0.902067723111, 0.547746633735, 0.158435508917, -0.208265848525, -0.628990277088, 0.572162738409, 0.091285246118, 0.383730288054, 0.903400742168, 0.899370619505, 0.409534416843, 0.721432036419, -0.171166404881, 0.037531974106, -0.923997071504, -0.113982760314, -0.780465516076, -0.697778906118, 0.818445268006, -0.590523809214, -0.171407635527, -0.610750438511, -0.662726470352, 0.271639270079, 0.430827816825, -0.113990542861, 0.717940707740, 0.748908513575, 0.136771315412, 0.820956531665, -0.827648688243, -0.863989622980, 0.510781040232, -0.902120915451, -0.807354979352, -0.349421748268, 0.635400432082, -0.484592911038, -0.334974188576, -0.625415861932, -0.571767841976, -0.465300639249, -0.877974358194, -0.295243416993, 0.744226620731, -0.179565886893, 0.207531340996, -0.366675890084, -0.149096543674, -0.117815700724, 0.428201432730, -0.223791727240, -0.374806082459, -0.996388861807, -0.079249452770, -0.509844081507, -0.045674891403, -0.440046273099, -0.482288649525, 0.214892790090, -0.035347344465, -0.179260400766, -0.678074715747, -0.440784613352, 0.695462715044, 0.799643546103, 0.121836725671, -0.525839633185, 0.541538631258, 0.042687636792, 0.657176601005, 0.400032534671, 0.390034269384, -0.114184467168, 0.994123486006, 0.464706416014, -0.894852671561, -0.267108894190, 0.402002424630, 0.160977296129, 0.145466358788, 0.976531073927, 0.056719064699, -0.108518014803, 0.248657955733, 0.642098807478, 0.882274575211, -0.075050234752, -0.387849389007, 0.617082980694, 0.668408355761, -0.990995438959, -0.796071114181, 0.934107014787, -0.282962962945, 0.914221612194, -0.454371406874, 0.420398416529, -0.665824266955, -0.618566845789, 0.831084959587, -0.534987119828, 0.461148218286, 0.306078529549, -0.151742796527, -0.026015973197, -0.157735142413, -0.339520290351, -0.931051734632, -0.365346093645, -0.002225437347, 0.232831108132, -0.177404032820, 0.882245684523, -0.954178340038, 0.274990354804, -0.399527887776, 0.358048197887, 0.673515953803, 0.518411076586, -0.415020034931, -0.299868827720, 0.047456389550, 0.214993655963, 0.268555680928, -0.968453108577, 0.257861939024, 0.379408565827, 0.965913300373, -0.875854620537, 0.402543694330, -0.538524422114, -0.875649232985, -0.863428966901, -0.882617351428, 0.375087296705, 0.673440480300, 0.292068266375, 0.644043062216, -0.380148068958, -0.859870226482, -0.686025308272, -0.555657058657, -0.340355923972, -0.657490223017, 0.568129117819, 0.872158742728, 0.670356628639, -0.477574660769, 0.817331344706, -0.679945936582, 0.915722789645, 0.046172274302, 0.637048459704, 0.820068547051, 0.613851939895, 0.523961727584, -0.231042052914, 0.685545054075, 0.038349575245, 0.401627308689, -0.165043382722, -0.476005923500, 0.181897513589, -0.509728059258, 0.711934265898, -0.110910195960, 0.135544444946, -0.203545678322, 0.121725756239, 0.667875415090, -0.662629857099, 0.534453835551, 0.073534356101, 0.955674602016, 0.716327577401, -0.505383061461, 0.201464649072, -0.255533045943, -0.628786980533, -0.588780931270, -0.186636679105, -0.899471910220, 0.637859966244, -0.685918583844, 0.751607301602, 0.823050845274, 0.874034840312, 0.350531785053, 0.364133563102, 0.417303337627, -0.759031868112, -0.159714839585, -0.572495224891, 0.683268462042, -0.476691720750, 0.867949662476, -0.986907373894, -0.195229753954, 0.446764162700, -0.007593856855, -0.385917986662, -0.999910422090, -0.288038894845, 0.247883233370, 0.499214163589, -0.979960644666, 0.409109548152, 0.604365030955, -0.752059503253, -0.098716987436, 0.261840857748, -0.310421840836, 0.273036546583, 0.966283042994, -0.512419815859, 0.223807017157, 0.204832588236, -0.126778911159, 0.559677233312, -0.312489754796, -0.130559768854, 0.344979245612, -0.995738541041, 0.850135154641, 0.859556583783, -0.543090391431, 0.363764893193, 0.863579500924, 0.416769655519, -0.716493357372, 0.165233723667, 0.879255846651, -0.719193755109, 0.827530877332, 0.296285159044, 0.257581488476, 0.429469163603, -0.296730775590, -0.247378135775, -0.475968969101, 0.156990696039, -0.110782913209, -0.397894591632, 0.928031296231, 0.820762403773, -0.777284120923, 0.829749477105, -0.225872893277, 0.521154183131, -0.448414615240, -0.107872120866, -0.839344971377, -0.477732735712, 0.067316773398, 0.269758615907, 0.052404674492, -0.967008085228, -0.077971909436, -0.832627790185, -0.897211929296, -0.750780680221, 0.148919714675, 0.064021695691, 0.427457969280, -0.064800288486, 0.247754925621, -0.612484958621, 0.875249801105, 0.647953509070, -0.259754750240, -0.368335454917, 0.636967637997, -0.656662520290, -0.097478340411, -0.837053812543, 0.527496448987, -0.501134811721, -0.031980809441, -0.889659422432, -0.729835289653, -0.403920662593, 0.911833319274, -0.195394608538, 0.579983597887, 0.480878402094, 0.753295698404, -0.886557102388, -0.481051881669, 0.858752026661, 0.419439422595, 0.424707540380, 0.070671397664, -0.607165311260, -0.423632073663, 0.067909420480, -0.598470181812, -0.525774866523, 0.950714625230, 0.599861469287, -0.442861591818, 0.069620972834, 0.541300442667, 0.327490730799, 0.309082582040, 0.047253630814, 0.606651953953, 0.112544392696, 0.218055864524, 0.106968569698, 0.599462743203, 0.023550831903, 0.337815059310, 0.932264427175, 0.165960823492, 0.733249781045, -0.789431880042, 0.493722751772, -0.004488036016, -0.691545281081, 0.051434132048, -0.767664479342, 0.141488503409, -0.281316569424, -0.517286821248, 0.770675414438, 0.853427796276, -0.657209527482, -0.742725530343, -0.427013088695, -0.483223026887, 0.856541610703, 0.723705297730, -0.817544392274, -0.863812634951, 0.190487237743, 0.462198474418, 0.038100294980, 0.386360398109, 0.138093633863, 0.668065694067, -0.322052819469, 0.694404971202, 0.497259150758, 0.048078271919, 0.614850342950, -0.443216140498, -0.793653679765, 0.901627621897, 0.311872553282, 0.787310048058, -0.793855935575, -0.913720147731, -0.322313905779, -0.139500835847, -0.031831499233, -0.199892750670, 0.779717894037, 0.221123175177, -0.472991991045, 0.820421631406, -0.784247416860, -0.382988401296, -0.862138590325, 0.423435170567, -0.804372214538, -0.876593305913, 0.414554638112, 0.690384876731, -0.460644141012, -0.473321310585, -0.262625983811, 0.898335619536, 0.260679529821, 0.275699048997, -0.994264328699, 0.602960163802, -0.216638281855, -0.490344920037, 0.737015766298, 0.221647194511, -0.352968279409, -0.134519186654, -0.273626093464, 0.709228485444, -0.663208857573, -0.757535911133, 0.918108741001, -0.942949058606, 0.684475031813, -0.682159656169, 0.044424281903, -0.681026442177, -0.550846721858, 0.680676646566, 0.115083908438, -0.475380034855, 0.031236674021, 0.309528795181, 0.396497086310, 0.992561703820, -0.828608440171, -0.662821048169, 0.345443857269, 0.511783158770, 0.701092811961, -0.154665388649, 0.857411359782, 0.807768488786, 0.176563276807, -0.262657388798, -0.537263630008, 0.327682125245, -0.195002137162, 0.416130858898, -0.466182630628, 0.440430297927, -0.558656953019, -0.133970113749, 0.877224542781, -0.640643669335, 0.175780660046, -0.147882721452, 0.214081434003, 0.055607726695, -0.504690715015, -0.647660320770, 0.141522624346, -0.709032275134, 0.560486701112, -0.692619269210, -0.323622492407, -0.856721228447, 0.538047401446, -0.385786684720, 0.497652128026, -0.608579764541, 0.046673550854, -0.524716032653, -0.513458687505, -0.802148264126, -0.718972019465, -0.809695136345, -0.174937573729, -0.459699622109, -0.431556777774, -0.377164596626, -0.653806773416, -0.495328156416, -0.376523729440, 0.669045504275, 0.687682292995, 0.409745264703, 0.409698822451, -0.314637937582, 0.421181934329, 0.426145288987, 0.411239972315, -0.143971067142, -0.472530929786, -0.999376532103, -0.010117384944, -0.252446404507, 0.568689736131, -0.384579797806, 0.105797046275, -0.986014968661, -0.358988842273, 0.463099585531, 0.579498127847, 0.174069383888, -0.294564146505, 0.383791518921, -0.352819525007, -0.751197789421, 0.238384371689, 0.575958789292, 0.325567966100, -0.775702038994, 0.586055162359, 0.015762489652, -0.790104117329, 0.105873643257, 0.411658492741, -0.348339320392, -0.982719945801, 0.548902146145, -0.825606404302, 0.197116056386, -0.658666172336, -0.964479301316, -0.818704439072, -0.644408803838, -0.578548088605, -0.925692159326, -0.228069188766, -0.662552251899, 0.145382647632, 0.410827400040, -0.097163171197, 0.524975835549, -0.545350325804, -0.924369765877, -0.871078875314, 0.640834814893, 0.745794714895, 0.645476673311, 0.816373640524, 0.660481824045, -0.019329983308, -0.174444134561, 0.008509437553, 0.718182955315, 0.421438827594, -0.589750350198, 0.863020074421, -0.534470850901, -0.487310067966, -0.046868309168, 0.118498474737, -0.567631551457, -0.893789349031, 0.111917085452, -0.780230280061, -0.653497496174, 0.517018493288, 0.220633771232, 0.459112770183, -0.928205266632, 0.656898353644, -0.483808580172, 0.547447574349, -0.674440746574, -0.610672731793, 0.927277458029, 0.825506128691, 0.248231844156, -0.478557259882, 0.670298284369, -0.043719508526, -0.290727658337, -0.361422090257, 0.948970050555, 0.571211060537, 0.331947663435, 0.391540362592, -0.168129930820, 0.788132594964, -0.458071788013, -0.057843938125, -0.615253173260, 0.299805842239, -0.802359906586, -0.271655375124, -0.583424020451, 0.247170669845, -0.089237113690, -0.955580797901, -0.691849111829, -0.625525753810, 0.334321355052, -0.210250415701, 0.975713460950, -0.551570788964, -0.735481025987, -0.576053802898, -0.437960036849, 0.322455075861, 0.309870803261, -0.316773385043, 0.928040673837, -0.121478860441, 0.936985092037, 0.334479511865, 0.077340483645, 0.804023797725, -0.260543885714, 0.352038790026, -0.673334760316, -0.577768216694, 0.092893685951, 0.211080078462, 0.404319179727, -0.249737852186, 0.752486932045, 0.162398853086, -0.901051886249, 0.486410134054, -0.979809914914, -0.198115550586, -0.007249442145, 0.797872230895, 0.997717591935, 0.732814017231, 0.892591137252, 0.498196079629, -0.815816982001, -0.050342233270, -0.521236123169, -0.349672510594, 0.132732176530, 0.892460200155, -0.751690695745, 0.645648352953, 0.295298566529, 0.596168128515, 0.753852190381, 0.775889617173, 0.599280300543, 0.768789926120, -0.095563371426, -0.973844451721, 0.524080710421, -0.376303503006, -0.485229695550, -0.858942355628, 0.500599253436, 0.039926936378, -0.449610628307, 0.124016399453, 0.555638716739, -0.498417758413, -0.420856983175, 0.999029911090, -0.961093982264, -0.738289444812, -0.085192780626, 0.391810947010, 0.516447957312, -0.639465369036, -0.837091914030, 0.699360516292, -0.198587431368, 0.082410681736, 0.765720099984, -0.177359173445, -0.031876021494, -0.479541180246, -0.740542530919, 0.957917378801, -0.948390493476, 0.866574505446, 0.093655648830, -0.944034261871, 0.773327126883, -0.574295769670, -0.518124168627, 0.293613250173, -0.597473245068, 0.755945496046, 0.933304784644, -0.333019192500, 0.383238400688, 0.526374353051, -0.853584808087, -0.738580426032, -0.331110505691, 0.524178678541, -0.495558182949, -0.899076756135, -0.015412120276, -0.092582756823, 0.697556773482, -0.499966619988, -0.036853902291, 0.879312708384, -0.109576945084, 0.009175009685, 0.099508293099, 0.136935455562, 0.392722695828, -0.420667048584, 0.607127244576, 0.984695379888, -0.163782934507, -0.549644422923, 0.513549503570, 0.925508393581, -0.255009979572, 0.609262841823, -0.021193500239, -0.541789592832, -0.613882790944, 0.902155639323, 0.678615981560, -0.461929508006, -0.084629200065, -0.273007190663, -0.711194393717, 0.499258514395, 0.625397679928, 0.664594211938, -0.263197178606, 0.620762842919, 0.882348542333, 0.928022772401, -0.334853145062, -0.154845691010, 0.863815493458, -0.829639009837, -0.182445739571, -0.906220219477, -0.561447714123, -0.769955136566, -0.594628431961, -0.292206696676, 0.618906581605, -0.439095465100, -0.366018131382, 0.407319088052, 0.732119312417, -0.735010247830, 0.678585596261, 0.339466473956, -0.881390338206, -0.736278151056, -0.889597356662, 0.541355736658, 0.316292775127, 0.148014392068, 0.223189988951, 0.479998607985, 0.330481521753, -0.223134566617, -0.190247914778, 0.281426168014, -0.296369895074, 0.718651766283, 0.869352765614, -0.207686781396, -0.782552643117, -0.651847670081, 0.455603345239, -0.488226839721, 0.163136971340, 0.800684569232, 0.858983058975, 0.751860753472, -0.358023298280, 0.325330482061, 0.809609122319, -0.760890582618, -0.928166736771, 0.656476871327, -0.937213106465, -0.921733664164, -0.475830893424, 0.508808172470, 0.255159840161, 0.259757582636, 0.705652729884, -0.087020950922, 0.976219451336, -0.355676086581, -0.936709635622, -0.979396294829, -0.898245320689, 0.596830327285, -0.217465147476, 0.228593853339, -0.788546553797, -0.896188841735, 0.710079375577, 0.834342165163, 0.194208097690, -0.889414160808, 0.627466473747, 0.448861767538, -0.889430622862, 0.729848135279, 0.232207840916, 0.678984740434, 0.513067189590, -0.364461172605, 0.900225308282, 0.898129693826, 0.388100392626, 0.675049186773, -0.496830148112, -0.246389044291, 0.422409485521, -0.069758471918, 0.282857299873, -0.097240820592, -0.713936274675, -0.411823071316, 0.572501368105, 0.389956703715, -0.758606826908, -0.127168931917, -0.850887781955, -0.554966871724, 0.894983424125, 0.185523938233, 0.693138358146, -0.197265191790, -0.203491160721, -0.972953478271, -0.776174524959, -0.789994922894, -0.302125475591, 0.366567086152, 0.696668458460, -0.262059911455, -0.091538051390, -0.174227813118, -0.521944029812, -0.639116745209, -0.994722702071, 0.248421896079, 0.733717564205, -0.441311340158, 0.768425722051, 0.520003199325, -0.639212138637, -0.180891064374, 0.519298301347, 0.180855598097, -0.612161679453, 0.754579307788, 0.960201120260, -0.476694950357, 0.637902991314, -0.883802242767, -0.406907694780, -0.698293447577, 0.363727624772, -0.551344329860, -0.789311971844, 0.611764313057, -0.933333158754, -0.816922461754, 0.152316955752, 0.478475923833, 0.955835157038, -0.992696367872, -0.215975653150, -0.596853601993, 0.175098734181, 0.291837294588, -0.349292385654, 0.491399179262, -0.353079439055, -0.590957321614, -0.874754887564, -0.961757632136, -0.930999458820, 0.283424173409, 0.520624351676, 0.008262324147, 0.020881745513, 0.744737608930, -0.679884618745, -0.831962244377, -0.840784651246, -0.560567109129, -0.642876168801, 0.311818897047, 0.101128681392, -0.638011814338, 0.872795850402, -0.159183999846, -0.904681946102, 0.354905173733, -0.515267683312, 0.581969072983, -0.127418089591, 0.230260937261, -0.741946939285, -0.200768179343, -0.980609810479, -0.684763731473, -0.516433875085, 0.986685959321, 0.470386428852, -0.872768208249, -0.558895352344, 0.149937150206, 0.615825539633, -0.264722417196, -0.377096516585, -0.856346137153, -0.788942459577, -0.870140315556, 0.163941326587, -0.404932474401, -0.086969831256, 0.275572447356, 0.130528653947, 0.225626064900, -0.300687807258, -0.063137772755, 0.413460969163, 0.430496368348, 0.374608436244, 0.110159988194, 0.383531273735, 0.026336885273, 0.481870944866, 0.572793544103, -0.841410923094, 0.726230130592, 0.422626465773, 0.987040902479, -0.752527232920, 0.337336279758, -0.274087008168, -0.005517808787, -0.921366596279, 0.916932265906, -0.497163751751, -0.155037225965, 0.310010659139, -0.566412550499, -0.275858488149, 0.510696795999, 0.823895828606, -0.598537121361, 0.481641736745, -0.435667888216, -0.412970162287, 0.453096732529, -0.750004660313, 0.121717794140, -0.720106880497, 0.432886094516, -0.074623212176, -0.020748418849, -0.078484791591, 0.636717008777, -0.067284118653, 0.375459220207, 0.124895765900, 0.230410446731, -0.902714563247, -0.001864722325, 0.937479300039, -0.131320027758, 0.841670010406, -0.968851784224, -0.184493168388, 0.905435162382, 0.692667741964, -0.317444067630, -0.722457782211, -0.739143464615, 0.035789919223, 0.068841841490, 0.511247473820, 0.322821098972, -0.212686382587, -0.007510391113, -0.487271832184, 0.949211182090, -0.307437882377, 0.449499244891, 0.162254494902, -0.306795679625, -0.010127440304, 0.747336956906, 0.142761180780, -0.640301590947, 0.531098984791, -0.857075049402, 0.663637731926, 0.817908313858, 0.878376984735, 0.797160005317, -0.408351772023, -0.784646267207, -0.780465634731, -0.676144467590, -0.610308003312, 0.844588028061, 0.829858125174, 0.643585446652, -0.426313608940, 0.399038497650, -0.164260528142, 0.997434039516, -0.641906502219, 0.208004147838, -0.440246526744, -0.603319814376, -0.697535413795, -0.915244348141, 0.023402903934, -0.615366330865, -0.949611352494, 0.563554375640, -0.871067117361, -0.832000580396, 0.897450898736, 0.126694941714, 0.027490221083, 0.495037617696, -0.836886933588, -0.536122764534, -0.369049545039, 0.180840357339, 0.578901094828, 0.173752573076, 0.952523280192, 0.685589076436, -0.588390745007, 0.584014422739, 0.389192578675, 0.805180913453, -0.837683150684, -0.535902970417, -0.795579368694, -0.672488921187, -0.401967403023, -0.266015411193, -0.700071656406, -0.661537605497, 0.428578951305, 0.307438231288, -0.319134311558, -0.158229865472, 0.122100948536, 0.316647537089, 0.654881180467, -0.601247643044, -0.285971434096, -0.120996636816, 0.307013345399, 0.024607912723, 0.780866321402, 0.827011782153, -0.408099091611, 0.278959308761, -0.324110908146, 0.954667413246, -0.994200123295, 0.733667119162, 0.982355521575, 0.585910600089, -0.245053104507, -0.869890049586, 0.390384356232, 0.055915341397, -0.494593369296, 0.067978157636, -0.209797929688, -0.234475593468, 0.097162281058, 0.870141800427, 0.096384253332, -0.952188287095, -0.731345573698, -0.165482635994, -0.187444199891, -0.591497502129, 0.332033942900, -0.690309656181, -0.396239220922, -0.156037720211, -0.215056180847, -0.769707059926, 0.675887223483, -0.906017205847, 0.876468187997, -0.708124183046, -0.281495100912, 0.776569334970, 0.857072888627, -0.809628008201, -0.079249219029, 0.406455587530, 0.627005649405, -0.155311231490, -0.857086400652, 0.274471601053, -0.930818098687, 0.007788139760, 0.465969417580, -0.416164815180, 0.992546790862, 0.993396258669, -0.012690712410, 0.938815587371, 0.010082268904, 0.333626233432, -0.946598206468, 0.023833684820, 0.755018710801, -0.583796230848, 0.744636654121, -0.054803308345, 0.119361100535, 0.904737230522, 0.105433415228, -0.100465796471, -0.400813965188, 0.986573964897, 0.960560568472, 0.343893558841, 0.321191542146, 0.591949840905, 0.203709843240, -0.089766909462, 0.659283434562, 0.834650680409, 0.599946686403, -0.893671061764, 0.185193125906, 0.598243851156, 0.494653358191, -0.824234498133, 0.330137485214, 0.459199718746, -0.380078786452, 0.621342974535, -0.201678517679, -0.585751577309, 0.352290586741, -0.669451432036, -0.218928073481, 0.058108217223, -0.031196588873, 0.092125031325, 0.346035679807, 0.623253353818, 0.833640879585, 0.090154576628, -0.377337664102, 0.558057164890, 0.281314752040, -0.033178260345, 0.759655753140, 0.133419436721, -0.007246190471, 0.375981724986, 0.185416510648, 0.445840061143, -0.598456736854, -0.273561798910, 0.635935834108, -0.671850717339, -0.183411776600, 0.656991651101, 0.282871652770, 0.685120867775, 0.166078367253, -0.264592070327, 0.542095741840, -0.519628703952, 0.500120307237, 0.741991020344, 0.255474688638, 0.918802912911, 0.199181168394, -0.594989788846, -0.571215380403, 0.608282066309, 0.460729143748, 0.833252717266, 0.084964647411, -0.370913351739, -0.363003122658, -0.925953646722, -0.782427060836, 0.846933504079, 0.285436644766, -0.143414031599, 0.668915138352, 0.898862442394, -0.437177081853, -0.179762632112, 0.483008894533, 0.574112519179, -0.282132247853, -0.671290005477, 0.182962117500, -0.500901080645, -0.131995091164, -0.008479864088, 0.570597108055, -0.522285784494, -0.698203600301, 0.567216683405, -0.253991031154, 0.198616690912, -0.206159691877, 0.874299254920, 0.916073463883, -0.177599802708, 0.052856943129, 0.321599342233, 0.487713571286, 0.434875109480, 0.454981547059, -0.447310547138, -0.751544863139, 0.257341399761, 0.738761982079, -0.915505782082, 0.918820821766, 0.489762818442, 0.108751866942, -0.142419326852, 0.045553815659, -0.053248908496, 0.564844001614, 0.576431440231, 0.197238681554, -0.554588211541, -0.896750490750, -0.107015089260, 0.757671946286, -0.988318593464, -0.285849613744, -0.070193964846, -0.866073238372, -0.131218499251, -0.542815144688, -0.192486590434, -0.104898053726, 0.403113899086, -0.350540387012, -0.915667517803, -0.332927497451, -0.335765375710, 0.038520578308, -0.143795935176, 0.441189786120, 0.650084443526, -0.656768821387, 0.723359834066, 0.828551591458, 0.308912870497, 0.676796020016, 0.065360105395, -0.922536305931, -0.348531898237, -0.513304823627, -0.297827637166, -0.082461528155, 0.016276713804, -0.786380409409, 0.678030100136, 0.147740819944, 0.176282510828, -0.431260850842, -0.132132095003, -0.413929670555, -0.005764474600, -0.330964537867, -0.100162800351, -0.472941169805, -0.542679986802, -0.874061105223, 0.100356010592, -0.463659755249, -0.278680910166, -0.542046476870, 0.552864273666, 0.468671758513, -0.124295035719, -0.460734974844, 0.668283199659, 0.927737905991, -0.167147762855, -0.277013105851, -0.923891595109, 0.906674795184, -0.455028116401, -0.540008041009, -0.494869166885, 0.526172181884, 0.109719054742, 0.081916195555, 0.388724821274, -0.476841311760, -0.937955600408, -0.595912447157, 0.832559243544, -0.899913786612, -0.276283055448, 0.506865544814, -0.407856026634, 0.615870788700, 0.275574874856, 0.450884058482, -0.913986586630, -0.349312684610, -0.030949128255, -0.719515909072, 0.665314379703, -0.154128193046, -0.371970584890, -0.621737057084, -0.723639193437, 0.950174798983, 0.003496887784, 0.863738081479, 0.063604209810, -0.344069899287, -0.837636455085, -0.277143252239, 0.179692395755, -0.399215308999, 0.650553170401, 0.047417792552, 0.053148296668, 0.659544150477, 0.432211420512, -0.281196656581, 0.667557712592, -0.671350631398, -0.236148780578, 0.956216656540, 0.817977570264, 0.427997328548, -0.155470437325, 0.519823354454, -0.268595554176, 0.006613729587, -0.803166393168, 0.305451800563, 0.625532453949, -0.611482469379, 0.041672018585, 0.175701108134, -0.932207163341, -0.570526755069, -0.182547074452, 0.208498231301, 0.361165944766, 0.413513154068, 0.401338295736, 0.407815956316, -0.467221204260, 0.644252080100, -0.091443607103, 0.957892815619, -0.440636580169, -0.387089664734, -0.493075638781, 0.641286876349, -0.028253600635, 0.580984483796, -0.692302690704, 0.113217917648, 0.090548988898, 0.285623446365, -0.913546296501, 0.288219985462, 0.615633782362, -0.778091071411, -0.431404256373, 0.909327872495, 0.827143535825, 0.545499754688, 0.134469798778, -0.669786232709, -0.937669371482, -0.558688270138, -0.116439050790, -0.372460446644, 0.555591598562, -0.960017793317, -0.746107610008, 0.511851771589, -0.365835468561, 0.707396975177, -0.019130076624, -0.602736726515, -0.458292025987, 0.315853928913, 0.385721257797, -0.175073250788, 0.485108885409, 0.263458181878, 0.282884209581, 0.252253570847, -0.885262243135, -0.901965958264, -0.586618336778, 0.586978002277, 0.956268688056, -0.026652825884, 0.526689044036, 0.084461592036, 0.992199164064, -0.046696321528, -0.204073634724, -0.572075186271, 0.667129135406, -0.557670840681, -0.623571944409, -0.127764794039, 0.677436036029, -0.243928992779, 0.115454645247, -0.106261316465, 0.875817640192, -0.911659216030, -0.723180445731, -0.749917607226, -0.143613217245, 0.510782846208, 0.592148535170, 0.755937850729, 0.143577208851, 0.748608641766, -0.047832373406, -0.277641989027, -0.393798066807, 0.906563806375, 0.236514075822, -0.654547536639, -0.547004015725, 0.319959414204, 0.810180401437, -0.492599210717, -0.642312728580, 0.563847564487, -0.429612325808, -0.905112594777, -0.952594002848, -0.346697424472, 0.583233488458, 0.073636746695, -0.136441075915, 0.082907096557, -0.305054636901, 0.285293010300, -0.893563847112, 0.322084070962, 0.971882025856, -0.146156755466, -0.356956540131, -0.746482271441, -0.309283733816, 0.651656064463, 0.375318446725, -0.431665101072, 0.619496901793, -0.702714202971, 0.213112447858, -0.454193434429, -0.076761482572, 0.977784305799, 0.275252647113, -0.846696395746, -0.797319732120, 0.372925045161, -0.772170292448, 0.640181446660, -0.380250960008, -0.287290543455, 0.224505263591, 0.011578759763, 0.944558001616, 0.806593283333, 0.515954696930, 0.084951472458, -0.316884986536, -0.864354010116, -0.003443897138, -0.690827655473, -0.008520744446, 0.220396687009, 0.200235831171, 0.685889373916, -0.014026315761, -0.787443790026, -0.907284922892, 0.939170388381, 0.925558380706, 0.161408122255, -0.044713406894, -0.394265986689, 0.379484965817, 0.014114186380, -0.623414619773, 0.817012000225, 0.255261319168, 0.135582969896, 0.338465737203, 0.442524817903, -0.466978297911, -0.168652193127, -0.151517063576, -0.358379111216, 0.643324049335, -0.085836757439, 0.340949770070, -0.245096435721, -0.799980577993, -0.764459273351, 0.467513495684, 0.783026918621, -0.637839056728, 0.445638069827, -0.263730123257, 0.010592797117, -0.679534831443, 0.021620059157, 0.194340703903, 0.113573130237, 0.784868487428, -0.149437997084, -0.204534660833, 0.927329646419, -0.644591449821, -0.852819168526, 0.473848525185, 0.126952720835, 0.899645866835, 0.893068661739, -0.319139968905, -0.018704087532, -0.988755218068, -0.944404487873, -0.658413493227, 0.120834469199, 0.602879864628, -0.776891717498, -0.062369291396, 0.873428958418, -0.784975379154, -0.846081915762, -0.142634809539, 0.931194504200, -0.313697070642, 0.305513351038, 0.257762908231, -0.927682360219, -0.098896303981, 0.874223085823, -0.537347706236, 0.803169888173, 0.488848844625, 0.382007913398, 0.964750985250, -0.758298724618, 0.537455786487, 0.107640861046, 0.544733170083, 0.868079577869, 0.948820240533, -0.216135578088, -0.698443512442, 0.523734529075, -0.833728868662, -0.238937528073, -0.965614216705, 0.974503056657, -0.449732043573, -0.816792244667, 0.473488661445, 0.538573132000, 0.927032186378, -0.015042549161, 0.900491473952, 0.744018480803, -0.160571460367, 0.347232615524, -0.740895859057, 0.597252212874, 0.398417747784, 0.232333936277, 0.649709894456, -0.925999495066, 0.208587663975, 0.022625988947, -0.717523335040, 0.528684482541, -0.675050725574, -0.935182112512, 0.885518136690, -0.482580827497, -0.307067575977, 0.804877435392, -0.612427297659, 0.540499277579, -0.233290650688, 0.844708915716, 0.721638564260, 0.425724541835, -0.047764247268, 0.109228099923, 0.165414523015, 0.515354846984, -0.230616510227, -0.908300957634, 0.254102263313, 0.822936386857, -0.981111321943, -0.448838948150, 0.201409773611, -0.852457498047, -0.150783730079, 0.119135940910, 0.466363007387, -0.291704000931, 0.479330580161, 0.118603936377, -0.880188072606, 0.073925932023, -0.721002649495, 0.392417577719, -0.367297090006, -0.991687012920, -0.759179923035, 0.680629086506, 0.949742642504, 0.184180501039, -0.419828691136, -0.375543736112, -0.087977990679, 0.882868370594, -0.841993230817, -0.016909588622, -0.220348526517, -0.707218413695, 0.886671984147, 0.450162741506, -0.473257665386, 0.579109903686, 0.877339078479, -0.466099698639, 0.900815725431, -0.152783389157, -0.171415998844, -0.039348570148, 0.377848623985, -0.805779856106, -0.449851139936, -0.814897092199, 0.228362750070, 0.461454696276, 0.293342659885, 0.232016631242, 0.449565200596, 0.472274598620, -0.497226065248, 0.882437907402, 0.962846404068, 0.464498807240, 0.299574037510, 0.776570521273, 0.850789179926, -0.020014049675, -0.731689246521, 0.979461939987, 0.226464561547, -0.233649210390, -0.641094679233, 0.024766801857, -0.293172355117, 0.785085278957, 0.454942424497, 0.964972364523, 0.900408833218, -0.359536150480, 0.657369721850, -0.827064837150, -0.362838484702, 0.446376467446, 0.371121470796, -0.882260863707, 0.132919901095, -0.364274091071, 0.487465099217, -0.923314610948, -0.081371798391, 0.404264394874, -0.016389056937, 0.109605946532, -0.673958412330, 0.494409078238, 0.966298249016, 0.827035024124, 0.127097863229, -0.324514234164, -0.524831997713, 0.079405087269, -0.702762926942, 0.671524413854, -0.142110193804, 0.313163514726, -0.380787058434, 0.939062407575, -0.222811623275, 0.871878070786, 0.586834825917, 0.428242631222, -0.252867501196, -0.728391979474, -0.685929931857, -0.330152198541, -0.913470155470, -0.323412732592, 0.152384301083, -0.137226454335, 0.011710722352, -0.485616713634, -0.530712319460, 0.492775637521, -0.698341234011, -0.326907646636, -0.958597046699, -0.066639077111, -0.167714051815, 0.476218846883, 0.149571477180, 0.342557107941, 0.732787920400, 0.989675160413, 0.078911521042, 0.229129997374, -0.761942924411, 0.356233143200, 0.270760062100, 0.149178685374, 0.057768049384, 0.406998598779, 0.240983473559, 0.446273008384, -0.911841372132, -0.292597426647, 0.681429406545, -0.236841997841, 0.746986228289, 0.537688475421, 0.903214575293, -0.290727659901, -0.110640312665, 0.620536061572, 0.906366742449, -0.850872945331, -0.770302079309, -0.912750957989, 0.393696510035, 0.430208799693, 0.273724014821, -0.478577465798, 0.436355144422, 0.048678087613, 0.311876495704, 0.012712681187, 0.631713425798, 0.124146170734, 0.467423646117, 0.074680473341, -0.826274147343, -0.350724885632, -0.794128254472, 0.510365557128, -0.677082979605, -0.087204314802, -0.255308251673, -0.810557274797, 0.686355573384, 0.692221858075, -0.201164101811, -0.553840495302, -0.505251508502, 0.638540479394, 0.270485497016, -0.604345699459, 0.919759855078, -0.214548911361, -0.383422532909, -0.403233902189, -0.632084352061, 0.727831321279, -0.859470761388, -0.996389499555, 0.318516847913, 0.505767405431, 0.667470337096, 0.221771086662, 0.119531231587, 0.518785945071, -0.882300806461, -0.792748369323, 0.274540220032, 0.321083339318, -0.113937139255, -0.266808028786, -0.123547324217, 0.018357484918, -0.792834907439, 0.068620229538, -0.932909837639, 0.463468334877, 0.423224235459, 0.708245969552, -0.432439149049, -0.954993507007, -0.079755048895, 0.627735084692, -0.301818358112, 0.850892273741, 0.861211044491, 0.900481852247, 0.788082568812, -0.029894677068, 0.495503330926, 0.954450837492, -0.594544804977, 0.632130224898, -0.902237796716, 0.534786607759, -0.825015833917, -0.190383041004, -0.071851186796, -0.608497673619, -0.547041916240, 0.245635476546, -0.721992642723, 0.964832210546, -0.479407087023, 0.457180592520, -0.257216906460, -0.612363247687, -0.013197415428, 0.061218368782, -0.050100803597, 0.071543431832, -0.910085160298, -0.249317855211, 0.103540378428, 0.004971809440, 0.877278903026, -0.209931646208, -0.491225631073, -0.185953466223, 0.621712192847, 0.609151795292, -0.945672379820, 0.572276518681, 0.674471076847, 0.241056751684, 0.843469987661, 0.293075080861, 0.323536613552, 0.026823295729, 0.458895226391, -0.416091819581, 0.711090179960, -0.518548507618, -0.863075125137, 0.542731993186, 0.283275880466, 0.057802475594, 0.393798874189, -0.807904472040, -0.274157324888, 0.226529976125, -0.128319582050, 0.937399845588, 0.162118856567, 0.538161819838, 0.720558555301, 0.334549538988, 0.002800291385, -0.976312832927, -0.949846113299, 0.128477232077, -0.136908801088, -0.441568609241, 0.227041799431, -0.230499473009, -0.508282724132, 0.314313008333, -0.201098263425, 0.378206207860, 0.734196426618, 0.381209757995, 0.868802917188, 0.759819174195, 0.474060775388, 0.373847609008, -0.496521326065, -0.856414676316, -0.507229172153, 0.938617284147, -0.802713866269, -0.462870603455, 0.082750749676, -0.066752254244, 0.108319544938, 0.929017040083, -0.136854055390, -0.790017998641, -0.377638306480, -0.200989409626, -0.604847031377, -0.781871108601, -0.956997914005, 0.365940004608, -0.342987182051, -0.966217942760, 0.234268700662, -0.697626641756, 0.485831142806, 0.963090395295, -0.829739063242, 0.112249628193, 0.245463406950, -0.821647586811, 0.217361860762, -0.763809146225, -0.309163967311, 0.163507253490, 0.387367520725, -0.094181239139, -0.263191353044, 0.180175964307, -0.945634492705, -0.414890079866, -0.521506150792, -0.515206933750, 0.033006615430, 0.446040424483, -0.030184432180, 0.304850284390, 0.181539292960, 0.967752229700, 0.091852792225, 0.650939614391, -0.712975275094, -0.173324740810, 0.929786365538, -0.321892983999, 0.379263339176, 0.048000886627, 0.208762092476, -0.782586002845, 0.137603412588, 0.416973637315, 0.385446104433, 0.670280845468, -0.437792634611, 0.032531706913, -0.111216284292, 0.324995085499, 0.093080304439, 0.022890102526, -0.325933220485, -0.155281725820, -0.781785629938, -0.657334999158, -0.110378168758, -0.531463055589, 0.703194506842, -0.832570684803, 0.569609597730, 0.936154550783, -0.033590230368, 0.364289334400, 0.028273243352, -0.136834036842, 0.752113078096, 0.842430949401, 0.863398298311, 0.700536798119, -0.283721602638, 0.604582581144, -0.944599923606, 0.362458634080, 0.085029119270, -0.604521543107, 0.208962538041, 0.506042107597, -0.539027826400, -0.730757295702, -0.366369243422, -0.903639276939, 0.848457550116, 0.093558489163, 0.955105090009, -0.725201341913, -0.153554498795, 0.957677107771, -0.336660455660, 0.330360718894, -0.348352327741, -0.857554505492, -0.250189618868, -0.425692415161, -0.958569911495, 0.153712208629, -0.176303743160, 0.813312034807, 0.513512675772, 0.425340483396, 0.212185696764, -0.682056679787, 0.338834910240, 0.234523830441, 0.054852624106, -0.653558004295, 0.881196743701, 0.655947844957, -0.322453219303, -0.905199545642, -0.562368205561, -0.214775678770, 0.108471359334, -0.394647671646, 0.101012748407, 0.020055781336, 0.720867221144, 0.134544966460, -0.855507903817, -0.136748828993, -0.020738967927, 0.348265064059, -0.615084510405, 0.305908419124, 0.458382782681, 0.850456055585, 0.325012268869, -0.416323617073, -0.313279006870, 0.536738186177, 0.524799823607, 0.084152192105, 0.468210614355, 0.215341458847, 0.975830482035, 0.519294923480, 0.602617722523, 0.545968867237, 0.398031513924, 0.193208632554, 0.312421048630, -0.719909889896, 0.687998615692, -0.330229139973, -0.353016706296, -0.904129835990, -0.654052091129, -0.337280349211, 0.424999366217, -0.722047337363, -0.279411466496, 0.940319707773, -0.756820189171, 0.746718915474, 0.351777640902, -0.028547395149, 0.968090470926, 0.987122393880, -0.583925685112, 0.383491722356, -0.471273857003, -0.918134670059, 0.855798298872, -0.224576282084, 0.116646596465, -0.307241301787, -0.435868657830, -0.346979407085, 0.248695206823, -0.192595572516, -0.723573622464, 0.196757443942, -0.006912538838, -0.704273807560, 0.506835396364, 0.270619442150, 0.465559683418, -0.923005522822, -0.864652414364, 0.055278991678, -0.058467359252, -0.810631224229, -0.694594336921, -0.198053336430, -0.861244500146, -0.271042050285, 0.315444779312, -0.900329142141, 0.589760805918, -0.143038310876, -0.697380622434, -0.805497443166, -0.130495868499, 0.489606449179, -0.991917840484, -0.372073367833, 0.232966979513, -0.611780373125, 0.122290896222, -0.294393946535, -0.637701139533, 0.016718116267, -0.327327665487, -0.228526147621, 0.789154893264, -0.264487560945, -0.319040493396, 0.355866477303, 0.693580651105, 0.798606473518, -0.494717028637, -0.236883292290, 0.658966375769, -0.055496873283, 0.140414701270, 0.335265429351, 0.407833570457, 0.012232639001, 0.056193156151, 0.534808651731, -0.662222526650, -0.134091876476, -0.996607192415, 0.524404259444, -0.423884817026, 0.566395952209, -0.320663147962, -0.593207270475, -0.719941971890, -0.721694318079, 0.993732160094, -0.154208569567, 0.239507679970, -0.889249487477, -0.520952829001, -0.633173906320, 0.667411179793, -0.137388569557, 0.563310475622, -0.065967165608, 0.646067033976, 0.827290016246, -0.577413865520, 0.854755796846, -0.708308889307, -0.758417568002, -0.881823578630, -0.239108771576, 0.039870578250, -0.178545188964, 0.015471568948, -0.550733395682, 0.791037018835, -0.015310884471, 0.072234905175, -0.006074686228, -0.698289949840, -0.159151027460, 0.124086117414, 0.992912361409, 0.350709448577, -0.694185796266, -0.161870897374, 0.289656072445, 0.533152594913, -0.342234874851, 0.083305973941, -0.360622404843, 0.376289815838, -0.082145104639, 0.899939089371, 0.771102003492, -0.763458706187, -0.431889685377, -0.724650973400, 0.202301621732, -0.016925019180, 0.978578045347, -0.296404922430, -0.402757487153, -0.958280704323, -0.212914514469, 0.528520706200, 0.162303234432, -0.709862230138, -0.054739724374, 0.423780918319, 0.674274670843, -0.499496952571, -0.668812593833, -0.036294765647, -0.038489677378, 0.283222228432, 0.466092742661, -0.831597150107, -0.965840046622, 0.877542398446, 0.732548495829, -0.333195374238, -0.243008153815, 0.958020442119, 0.191080658374, 0.378617965473, 0.373289008222, -0.219368889408, -0.713296003847, -0.649794622248, 0.366869121153, 0.752212055106, 0.174689165409, -0.511527990240, -0.680534817039, 0.950461032530, 0.257668179428, 0.123602813662, -0.444889398577, -0.280014704540, -0.576220149829, 0.662755158177, -0.728011483579, -0.264928522499, -0.179003307151, 0.828667644011, 0.703398291745, -0.897565568702, -0.480217300915, -0.596815963119, 0.708558718363, 0.431843016074, -0.414010509369, -0.230674341901, -0.816111350114, -0.779680802547, 0.349884693411, -0.631284757269, -0.343238246356, -0.830531660023, -0.344846422321, -0.824111134483, 0.355283689059, 0.553766691029, 0.300558226735, -0.562329783290, -0.607258952405, -0.421276292985, 0.438849726713, 0.083049493590, 0.432347607886, -0.858819560250, -0.000696973725, -0.809514807710, -0.555239420776, -0.612835599233, 0.109485825383, -0.416104597498, 0.002912307143, 0.166457467678, 0.874324949958, -0.350108602581, 0.257271928782, -0.861939741186, -0.320314075783, -0.115617533699, -0.920852555096, 0.553351359988, 0.098576573857, 0.511207577733, -0.061825562414, -0.936799292246, 0.974547343396, 0.260010262121, 0.696945344713, -0.113926447224, 0.517583369463, 0.714681450414, 0.450333476326, 0.998582156302, -0.667934255839, -0.274174480550, 0.197717829566, -0.766396312427, 0.974453685294, 0.345606057914, 0.914001288445, 0.044460966309, -0.448682999617, -0.206657982433, -0.198701035035, -0.579644224064, -0.610740429503, -0.002413837441, -0.002898632492, 0.321205948304, -0.143399079157, -0.535104658816, 0.806840946321, 0.844192399109, -0.240344848557, -0.685207969148, -0.068479361574, 0.237107177045, 0.913322885474, 0.052040512469, -0.516489487462, -0.534736295378, -0.108354598241, -0.589801894592, -0.741230990795, -0.125467214902, -0.975355771689, -0.267728779654, -0.714016210073, 0.522298442580, -0.578884222933, -0.076890446514, 0.264061431902, -0.910988136972, -0.503324546236, -0.353109890207, 0.192689706821, -0.515938988506, 0.196865192142, -0.983223057273, -0.271433545112, 0.959052720418, 0.161656440506, 0.914539414493, 0.895568603002, -0.767443660210, 0.257605926448, 0.090927808330, -0.325520056005, 0.179929313756, -0.363646605889, 0.853606953320, -0.260474915531, -0.542089791426, 0.671635574772, 0.536708207748, -0.449571552826, 0.958953782558, -0.312667373016, -0.009837495224, 0.878541246376, 0.539559039893, -0.573454401716, -0.642701236360, -0.291531762667, -0.305889372373, -0.692290749167, 0.131319347674, 0.707610960293, -0.590992623148, 0.716937760172, 0.904295489437, 0.103830443686, -0.244015890933, 0.664116162558, 0.763263816782, -0.198235735303, 0.415020132728, -0.315518829771, -0.510990912905, 0.023295416190, -0.123186525714, -0.013852355164, 0.818854527231, 0.104017372911, -0.925849479204, -0.765659930650, 0.801516750045, 0.907342765007, -0.669464798234, 0.410619118928, -0.441244689712, 0.212252488156, 0.686280536095, -0.085694554235, 0.501830165029, 0.837405591594, -0.760738477222, 0.980269720710, -0.188465431238, -0.688004294936, -0.650455441742, -0.239280711543, 0.300155568290, 0.522179375999, -0.615750152129, -0.936590672919, -0.390643816641, 0.309759655237, -0.210155660853, -0.871910963229, -0.551146245920, -0.430517928562, -0.824923933437, -0.108776505941, -0.617251542016, -0.008269066614, 0.522881386049, 0.743435800860, 0.047571439195, -0.304459274799, -0.722959610262, -0.606529112314, 0.383833628521, 0.867434184632, -0.232466395399, -0.331007508611, -0.515817489967, 0.765237758615, 0.613400700581, 0.932040216143, -0.121716861670, -0.917156529496, -0.205325730469, 0.892578679097, -0.128108142996, -0.211553291846, 0.724230277478, 0.236513243265, -0.230644698479, 0.827260950152, -0.941544657157, -0.881030877804, 0.819110698757, -0.947705941322, 0.358607520501, 0.652392906781, 0.594452874619, 0.969914441406, -0.782608404028, 0.648193471523, -0.454356817368, -0.989563788188, 0.448633970764, 0.864379467386, 0.803420190766, -0.494606649011, 0.880918053209, 0.869387409066, 0.396251061612, -0.294080232061, 0.131713173370, 0.290240201331, 0.992785459585, 0.494884406929, -0.019086663937, 0.065075282533, 0.352423275158, -0.394250776364, 0.600535114806, -0.017867616290, 0.740860681248, 0.576131335248, 0.913362683331, 0.170894318528, -0.216437213364, 0.621176380379, -0.929104947346, -0.239952900144, 0.094437466794, -0.910744748150, 0.729675459182, 0.740217069187, 0.027831964543, 0.920153530432, 0.763206713446, 0.617760088600, -0.022411773381, -0.282189439350, -0.071664720501, -0.044129499416, 0.304636196792, -0.955078931406, -0.575710136362, -0.677483645910, -0.671639528430, -0.496266623105, 0.235455781257, 0.732466454536, 0.296783490403, 0.598403813835, -0.945436379819, 0.314891685327, 0.322395083401, -0.242914869722, 0.220017006708, 0.986613670751, 0.117783686625, -0.127854941093, 0.762046311144, -0.237982525507, -0.894829017674, 0.103652471035, -0.084755955441, 0.168174092791, 0.685386093816, 0.276986083190, 0.304302608029, -0.057348483868, 0.244927747022, 0.224406646898, -0.636194655838, -0.807993995024, 0.924926198938, -0.847521314959, -0.211921063857, 0.577117577143, -0.803554649138, 0.508916367746, -0.571267229815, -0.734869332036, 0.571575873837, 0.486181158176, -0.604089167817, 0.405666085940, -0.460729251401, -0.720930911542, -0.525315286359, -0.640354177342, -0.345107121595, -0.656326065605, -0.003515468237, -0.084310294509, -0.915112139860, -0.467345078578, 0.705618536507, -0.217498248625, 0.548854153860, -0.317080310442, -0.234852130222, -0.525494421052, 0.387647191499, -0.550212844940, 0.962629672335, -0.577042819825, 0.823481390841, -0.361408757199, 0.314044267506, 0.607699839174, 0.326229593424, -0.337132233149, -0.557776638807, 0.056044384431, 0.936186258734, 0.163767348788, -0.854951302673, -0.200970197924, 0.491085173144, 0.574075450177, 0.051948272903, 0.442307191573, 0.001858848234, -0.389212016780, 0.343956920581, -0.702959256812, 0.992085669208, 0.026883419149, 0.054251610730, -0.135172094990, 0.498048068987, 0.523829107038, -0.404965680971, 0.926650271623, -0.091340377604, -0.448310143581, -0.875544273451, 0.024705157381, 0.400066467200, 0.623962293200, -0.630093563474, 0.281266266709, -0.390491561123, 0.367854673016, -0.207430501876, 0.329597605797, -0.438854524306, 0.013959842098, -0.081836518770, -0.021444851293, -0.472736268602, -0.943199422059, -0.946357250678, 0.064993255235, 0.002892192232, 0.955235093091, 0.567259731091, -0.685500133935, -0.365737207900, 0.619055976551, 0.910520303116, -0.866765432412, 0.434907459942, -0.913304560848, 0.899152210173, 0.396019705571, -0.215220562145, -0.746301706790, -0.457672183158, -0.577382617805, 0.446021976503, 0.386595976653, 0.952894186554, 0.752019434364, 0.216605197329, 0.115791385262, 0.436287142227, -0.454230250267, 0.751526120711, -0.218272222872, -0.800913016963, -0.506216665506, -0.094145285742, 0.237290567629, 0.906398569638, -0.065219933341, -0.740921323494, 0.565216601432, -0.002623854807, 0.026482021759, -0.338563751678, 0.292334990860, -0.071287080514, -0.451744055325, -0.870921696692, 0.873729538475, 0.886847036744, -0.475129600857, 0.588259309305, 0.656114517526, 0.221753535163, -0.049786030852, 0.304819594707, -0.165678043221, -0.433761271382, 0.694013062550, 0.042534698489, -0.399959874872, -0.564147306531, 0.458681516563, 0.734831515327, 0.065201332298, -0.787916049709, -0.877631366329, 0.356870074535, -0.290003457047, -0.745931537381, 0.318131514151, -0.838921910082, 0.268395148094, -0.821248724096, -0.806080032724, 0.144155231429, -0.767837525487, -0.468545243314, 0.090066683387, -0.100797091503, 0.342748488415, -0.276925658913, 0.843618365864, -0.539942436884, 0.860192733634, -0.463556928127, 0.784170742668, -0.474960636576, -0.797323740038, 0.460947294754, 0.158280629113, 0.514940333765, -0.773900881396, 0.290730138520, 0.574082578867, -0.211923361495, -0.570438101222, 0.330663467954, 0.716216335346, -0.144942511232, 0.394272393983, 0.719840579169, 0.001629415965, 0.536038110333, 0.274521481674, 0.465054397805, 0.367302666782, 0.659652592374, 0.305096535944, 0.434685422449, 0.158233724586, 0.723718502693, -0.614692786942, 0.954473486403, -0.318711721361, 0.023523817566, 0.112032743349, 0.218760801588, 0.396378471911, -0.286337073343, 0.015039056482, 0.100302991576, 0.580292158639, -0.979792368387, -0.812317168519, 0.106806013016, -0.076008885537, -0.885917241967, 0.530251708555, 0.404272812810, 0.409508500405, -0.256980526059, -0.177432544941, 0.807934454300, -0.995694329107, -0.054756518272, -0.852065957830, 0.112815952271, 0.706960942788, 0.037657671418, -0.381931287408, -0.538015474209, 0.058901901475, 0.883511863798, 0.186329873508, -0.882814571517, 0.842160978763, 0.423888478526, 0.457585568228, 0.581464521992, 0.447936412906, -0.321643446678, -0.956050781519, 0.556387145722, -0.513693511507, -0.701452986366, -0.200415242720, -0.117217303658, 0.488402634357, 0.089341673839, 0.792561607868, -0.166443625142, 0.895505789323, 0.968577572768, -0.240290835007, -0.855501362480, -0.292379307206, -0.589258039867, -0.521457573957, -0.760683306875, 0.060168481430, 0.893441481245, -0.259926963876, -0.552041428568, -0.477954458271, -0.012584226773, 0.092565616102, -0.183858339852, 0.789928401465, 0.747444309944, -0.671573611815, -0.270246404978, -0.200496458335, -0.726702201596, -0.008015149660, -0.059532136024, -0.408250103694, 0.856941801357, 0.960445271929, -0.079203577733, -0.120235654682, 0.161523640637, -0.728040961404, -0.944728961700, 0.340305222854, -0.118671574131, -0.070989013238, 0.601852010502, 0.875009638863, 0.496113356178, 0.361426388432, 0.657063689224, -0.990705682242, -0.568911039501, 0.910409838859, -0.357496136399, 0.868234716287, 0.848408484427, 0.242461942025, -0.463422415336, 0.740711822598, -0.677811212913, -0.695973348381, 0.728504690527, -0.232766644006, -0.014677102694, 0.648244777755, -0.957929951727, 0.386948897714, 0.997808412440, -0.182235363707, 0.486351233443, 0.757627660144, 0.075813675663, 0.685105165781, -0.345706751801, 0.084442793776, 0.683072485474, 0.822610017990, 0.454593680450, -0.885888861694, -0.621647637694, -0.182365117124, 0.076245540246, -0.983395169168, -0.389122213158, 0.813777791190, 0.493129503398, -0.286525952348, -0.616048495835, 0.685360204940, -0.164441253143, 0.741169954574, -0.398275980331, -0.846205347050, -0.401880099011, 0.084532478985, 0.133908231596, 0.950224930579, 0.529542656643, -0.590850851955, -0.198740371041, -0.932357710567, -0.956692199955, 0.722090962312, -0.474970689473, 0.551809428203, -0.448843928931, 0.698335854946, -0.672125849739, 0.533213469402, -0.780822360663, -0.809194455325, -0.493511499002, 0.596564745126, 0.296424246165, 0.489499271450, -0.878005040562, -0.743350703756, 0.756053845197, -0.007591093796, 0.952102147098, -0.531099488591, -0.183647766608, -0.512568487806, 0.889724336892, -0.090612471202, 0.438713233472, -0.800806077303, 0.172386057336, 0.410763537054, -0.593854022499, -0.143041582089, 0.640687229533, 0.382218151751, -0.767283257234, 0.271574343593, -0.891079819002, 0.248972484285, 0.088327958751, -0.229636100065, -0.263360615166, 0.747104702024, 0.490979553498, 0.839052011794, -0.297972610625, 0.099610320045, 0.042257188086, -0.786098405823, 0.816745315563, 0.593381315087, 0.730912690473, -0.796580952124, -0.778140439759, -0.890111117335, -0.214253791949, 0.366751449835, 0.811608365793, 0.179657343598, -0.612135186160, -0.239679196084, 0.371109104911, 0.902585611134, 0.387826372623, 0.452716540571, 0.923325872420, -0.026699461483, -0.474534075520, -0.596462338438, 0.018166292258, 0.431979610468, -0.417896064269, 0.429677626319, -0.027974370838, 0.642801312738, -0.331749742473, 0.195751000764, 0.471457236876, -0.931383246314, 0.584985017828, -0.066107240640, -0.565602737621, 0.297285814811, -0.251422168853, 0.734850520612, 0.440594564464, -0.429238751785, -0.960420585671, -0.063452642151, 0.357114823603, 0.459659617108, 0.189293173309, -0.105560992003, -0.942622790999, 0.650022998675, -0.088802367207, -0.949111763531, 0.095815950170, 0.054666887534, -0.055911141737, -0.709542264445, 0.619983381652, 0.396765749823, -0.473541769009, 0.493955521807, -0.632996261581, -0.394304305316, -0.714984300386, 0.739333285290, 0.914359835892, -0.424240963928, -0.938880680149, -0.458567659387, -0.543973210504, -0.540794284992, 0.269982022510, -0.849085424959, 0.127005665105, 0.489162566596, -0.319191815522, -0.046173654031, -0.964700425158, 0.297952891106, 0.655675993312, 0.989106672333, 0.235190964697, 0.805482395664, -0.926792201668, -0.740812451689, -0.140065346532, -0.827768335471, -0.232991422452, 0.597856914576, -0.714942820756, 0.128244108872, -0.013202650030, 0.235114988909, 0.426038164912, -0.472484178250, -0.356093262087, 0.934303104322, 0.366389223551, 0.815899658030, 0.698272555227, -0.984408083497, 0.180266011494, 0.997781488310, -0.563527630115, 0.240980985280, 0.322053832133, -0.952492831850, -0.677327985708, 0.815932477702, -0.463103762441, -0.272040423027, -0.758693562523, -0.651412424285, -0.233727287413, 0.886831600919, -0.018580340936, 0.235064872101, -0.334760835380, 0.055435194353, -0.782461476099, 0.725801005703, 0.631260774873, 0.614879620606, -0.613248057440, -0.056038621275, -0.995946702355, 0.864628696311, -0.329785685090, 0.216509375617, 0.151901015009, -0.062665209589, -0.660805358746, 0.569187652987, 0.003997032125, -0.104143415997, -0.369007418982, 0.535058228078, 0.193913152444, -0.830640435343, 0.200375817167, -0.418082629498, 0.506901173588, 0.152024046264, -0.461997852583, 0.099763147350, -0.754029320263, 0.698131345050, -0.649772591333, 0.878770740125, -0.340537533269, -0.551791266589, 0.068145313237, -0.370842731057, -0.206098940077, 0.716768151615, 0.961585881254, 0.229921519281, -0.508266200123, -0.229152912036, -0.681576245812, -0.649080344526, -0.854121101650, 0.914429257322, 0.718882809691, 0.560349559892, -0.834244727228, -0.617731444777, -0.900166117143, 0.166674006167, -0.684986328410, 0.734241628998, 0.734908848633, -0.341116395412, 0.528429018733, 0.585722491300, 0.854084982600, -0.367027637662, -0.822121173112, 0.475120350276, -0.154657858182, 0.863087030487, -0.855231344989, -0.492136986635, -0.736728452139, 0.042235609238, 0.471710990455, -0.238747645870, 0.677766256571, 0.935646333012, 0.528330385998, 0.176331532400, -0.423273976287, 0.925535920903, -0.998847195460, 0.848041264252, -0.204956890132, -0.375374319774, -0.011692401407, -0.508911167928, -0.555524124916, -0.999128411380, -0.515175819798, 0.712474508305, -0.085466924582, -0.995767401621, 0.328574320347, -0.711169976460, 0.342869970514, 0.618256776782, -0.410172233458, 0.168885729734, 0.699281598589, 0.005798891779, -0.350695486080, 0.602020220917, 0.275478802772, -0.659642188283, 0.984724236670, -0.741781526572, -0.366081260364, -0.649978911632, -0.347484182558, 0.826039014089, 0.202731521537, -0.422289743504, 0.702487680528, -0.184249401361, -0.766032660047, -0.215251078097, -0.158074792968, 0.205593419734, 0.197617941957, -0.668078700440, 0.831654632222, -0.274184527946, -0.421134967140, 0.268923677815, 0.593243607717, 0.450615754051, 0.627867058745, 0.253295747797, 0.627152754491, -0.362757089717, -0.990149890152, -0.100604715349, 0.386754093305, -0.662054791310, 0.513081364737, 0.097592968375, 0.332364342293, 0.275034392925, 0.654285284272, -0.113302360477, 0.693894628347, 0.132837656652, 0.969935812696, -0.840442107137, 0.422182536889, -0.974967834153, -0.130477370216, -0.861958694980, -0.285731040018, -0.017798691107, -0.049776687282, 0.801647604516, -0.476942412385, -0.802431326520, -0.843275154818, -0.265419953695, -0.716755860256, 0.748535433008, -0.672488068256, -0.530650313774, -0.634590236755, 0.453320042507, 0.284180566509, 0.374274141570, 0.228011115307, 0.489802466166, -0.628637747681, 0.448479292187, -0.162771381214, 0.974968368383, 0.894428945020, -0.387238083279, 0.765138804885, 0.237770685288, 0.562598410404, 0.240477697201, -0.858613802144, 0.197982369284, 0.810155040636, 0.352625635055, -0.247914680837, 0.335681132928, -0.517014554492, -0.067681107965, -0.665929960551, -0.708793237407, 0.891652477222, 0.267258783683, -0.531562284109, 0.192263654698, -0.842098422346, 0.803104574110, -0.212533076898, 0.998224172552, -0.628688730222, -0.612442135443, 0.136603803506, -0.337700720177, -0.499263353756, -0.203612698016, 0.875118699275, 0.971677253049, 0.733117405548, -0.257113262748, 0.552901147235, -0.023996232154, -0.262927530664, 0.804442568630, -0.903592135185, 0.832457558286, -0.764756618015, -0.117219897513, -0.036340244348, 0.797326755204, 0.090348158565, -0.456386411855, -0.735141262810, 0.180943439135, 0.215971844119, -0.142633455816, 0.662788769005, 0.480783795293, -0.190263636756, 0.874108847438, 0.411421414555, -0.846868384819, 0.501748356417, -0.746322616528, -0.792334753046, 0.077445271633, -0.779728435468, 0.612523616127, 0.794643428586, -0.698707492114, 0.787221669917, -0.099620663199, 0.089094140918, -0.950929011187, 0.892466448745, -0.414877557357, 0.442032695515, -0.178502240818, -0.372202262295, -0.955546340019, 0.515181084997, 0.810031576455, -0.768656426054, 0.759655214750, -0.105755700456, 0.758239959087, -0.952995393122, 0.845829979627, 0.854279200308, 0.288330603188, 0.099955065073, 0.518530164563, 0.016458246944, 0.410399095084, -0.820370315169, 0.412419423998, -0.831132485939, 0.775123275388, 0.698297531403, 0.263834432846, 0.645364827833, -0.289725374569, -0.061659514585, 0.540821176511, -0.477179404570, -0.331626332333, 0.835570196918, -0.408115239492, -0.627669496820, -0.849071309937, -0.694345767125, -0.830008380435, -0.007065023274, 0.011950331027, 0.767984997922, -0.566543209527, -0.066219937213, -0.230560669104, -0.379636029829, -0.027071439313, 0.858259051579, 0.859592927680, -0.841600767857, -0.606142690339, -0.141266325008, -0.678860877800, -0.217578378293, -0.970511007981, -0.291073982436, 0.999708579227, -0.332997771368, -0.600867899174, 0.336350598239, -0.599897457672, 0.484497671396, -0.917366527917, -0.894033976091, 0.079941800418, 0.902937680868, 0.932763966597, 0.349037360823, -0.593017743787, 0.792917788166, 0.374521612180, 0.480803969249, -0.246129258321, 0.246604081990, -0.793102178900, -0.467213530494, 0.134788113889, -0.748302328385, -0.662320379672, 0.813877264670, -0.226499788181, 0.864242887885, 0.632761191267, 0.794265030101, 0.515802184938, 0.929914743348, -0.105197426205, -0.127221302530, -0.088851145614, -0.382447869264, -0.948521693886, 0.625450412344, -0.147214247587, -0.997754665437, 0.690629195083, -0.201011122308, -0.910471202259, -0.933043110888, 0.912393836862, -0.647813991644, 0.010939625943, -0.375415318419, 0.788652389085, 0.299403109941, -0.066326909133, -0.550220132446, 0.008669094380, 0.252240491629, -0.159181417883, -0.115447503554, 0.816130126579, -0.800964705769, -0.393519793894, 0.492723262518, 0.656351133568, 0.909674492870, 0.728540643889, 0.955729991359, 0.753181064490, 0.596754943938, 0.649046980094, -0.597979680388, -0.821709849982, 0.309326899602, 0.698191767806, 0.173793745644, 0.055925059893, -0.366946887899, -0.017327039012, -0.924209925924, 0.709520095693, 0.016985188376, -0.236463340961, -0.454308456990, -0.605894533562, 0.683610799853, -0.361272173189, 0.553484911721, -0.065624390049, -0.530772611725, -0.115232457196, 0.712518512226, 0.644864103193, 0.949708576093, 0.699930298897, -0.544763374629, 0.259345529289, -0.088216392661, -0.370315395068, -0.491032188247, -0.869706434353, 0.245227566000, 0.550663603751, -0.810291555439, -0.544137943482, -0.523493585890, -0.462561309212, 0.338623301615, -0.990521968142, 0.860908197707, -0.792750196393, 0.801172282122, -0.204966806662, -0.056788944519, -0.792258921489, 0.336271235013, 0.768914379233, -0.614510171288, 0.285356212282, 0.273607878217, -0.984249019657, -0.968245519674, -0.402489652431, -0.878184406609, 0.266972161010, -0.244205443633, -0.228177751703, 0.893685111902, 0.315803804965, -0.946602809267, 0.207214370650, -0.367676910298, -0.253446034303, -0.435892648684, -0.364361017188, 0.544229464209, 0.474146699883, -0.997761983320, -0.388631824973, 0.095759358380, -0.174712739546, -0.337231660613, 0.326948316924, 0.467794207516, -0.535100284302, 0.250753967176, -0.474128691423, -0.519723725440, -0.467284817843, 0.026636502142, -0.569738381829, 0.403538870746, 0.244776087675, 0.489157792977, 0.074210491813, 0.974823998069, 0.796177091063, 0.398040389024, 0.257283813913, -0.311760913102, -0.726436985437, -0.735123677915, -0.211841468481, -0.096971916562, 0.476440265482, 0.870926192482, -0.958831029961, 0.081387069227, -0.037000263370, 0.198357151077, -0.178652934006, -0.419908459336, 0.335407919144, 0.711243617198, 0.518790009240, -0.878675988736, 0.193735767457, 0.730618590569, 0.917680616826, 0.079874158826, -0.078480712241, 0.448450045456, 0.579173401463, 0.661990523995, -0.109615949852, -0.527556604869, -0.793986162262, 0.442723400484, 0.414376752543, -0.763178528518, 0.502000530954, 0.627613883547, 0.021552914532, -0.884074749670, -0.439331508987, 0.353202912139, -0.518118065337, 0.108598528642, 0.048001263114, 0.225994349137, 0.932909752040, 0.501169689417, -0.717334133865, -0.560373840097, -0.294955775931, 0.031556485157, 0.064753680813, -0.421698711338, 0.445055267573, 0.359476148168, 0.138322573588, -0.973385434859, 0.682470199393, -0.075017897780, -0.960942480894, -0.909105625034, -0.763927363118, 0.903620758776, -0.323153488853, -0.733016359498, -0.210744205904, -0.550325422761, 0.647841653392, -0.227386695007, -0.318045258493, -0.303619276125, 0.883039278738, -0.947022160239, -0.267679455187, -0.325998157281, -0.472233345856, -0.872909818369, 0.699870056113, 0.712854954610, 0.297538228844, -0.586435288120, -0.804113518928, 0.236713529132, 0.878974245712, -0.928247161878, 0.678530490019, -0.356755885108, -0.783369502047, 0.337065301018, -0.656643770081, 0.738992021428, 0.649035185235, -0.139419840538, -0.724712957360, -0.466756632325, 0.569859889254, -0.920728229592, -0.283376038782, 0.504927150058, -0.710069337219, -0.905705239906, 0.120736402129, 0.933865217558, 0.190131275064, -0.869894135682, -0.275937491922, 0.430504557886, 0.796200486518, 0.991970223927, -0.270304474757, -0.422013519199, -0.674436057694, -0.232959644542, 0.399189221611, -0.884811208288, 0.418274439340, -0.345412134434, -0.225132871429, -0.764096482308, -0.593808994071, 0.309758482609, 0.972479329996, -0.563017471022, 0.638189360252, 0.902387109896, -0.887379907063, 0.109829046366, -0.712584772354, -0.080974748098, -0.439476577255, -0.249009559610, -0.836453989173, -0.020933148993, -0.511647145914, 0.786638208379, -0.851363778740, 0.340673273278, -0.036136960868, 0.628328272071, -0.370510846323, 0.564114587658, 0.049372496962, 0.606415175666, 0.772330505167, 0.196018578641, -0.653014579082, -0.146296268749, -0.967081135646, -0.141457966110, 0.911344289187, -0.000253138025, -0.435897722906, 0.484552093532, -0.419671965822, 0.110604930283, -0.622637107323, 0.495477033211, -0.553481350726, 0.747946834845, -0.826943919401, 0.497251551066, -0.401620521519, -0.938073500120, 0.906415515039, 0.508398742032, -0.961334204037, -0.584025197814, -0.479559789196, 0.120493312005, 0.652018456672, -0.473317540724, 0.607886503889, 0.503916570789, -0.777530408023, -0.517480881308, -0.118068963776, -0.644327693660, -0.876453388056, -0.581995089769, -0.772654881179, -0.132136750652, -0.429625722430, -0.164121727420, -0.141558239411, 0.191335245853, 0.991994278740, -0.582965631643, 0.618537496395, -0.524636844792, 0.070740727788, 0.439975324587, 0.013361886570, -0.343175751297, 0.218920424829, -0.837908911382, 0.352202475564, 0.414187759428, -0.307443103864, 0.923663394443, -0.282888436498, 0.714945497387, 0.502538034398, 0.805664187816, 0.600573778359, -0.944674029633, 0.764132883180, 0.436425765501, -0.557699649458, -0.283251051715, 0.807858399194, -0.979584461583, -0.231545205021, -0.011616961202, 0.104900069062, 0.079618120056, -0.208823457736, -0.847430246301, -0.101013145879, -0.772975920986, 0.439345867598, -0.775191381780, -0.488486649505, -0.414832701277, -0.928578881809, 0.139656839902, -0.399947921869, -0.856496397700, -0.169955077039, -0.194557779782, 0.972119543076, 0.263518680911, -0.535249191711, 0.007957553010, -0.098182740396, -0.046496905020, 0.402313735176, -0.254053768397, -0.166833265563, -0.689194191164, 0.981559739720, -0.658191711640, 0.220090878105, 0.983495208841, -0.207876695831, -0.619503363950, 0.176334718098, 0.599918277710, -0.999776694870, -0.933859255366, -0.263611878547, 0.072453246998, 0.225805263444, -0.243509844473, 0.811662829082, 0.406614176621, 0.636469589208, 0.066219649932, -0.452009499960, -0.657494301943, -0.272170526523, -0.662925281630, -0.389661051223, -0.819754576452, -0.811646534904, -0.004885251486, -0.972838786638, 0.227047075182, -0.675657784005, 0.257759752734, 0.074758500518, 0.614049800094, -0.956600927354, -0.662138285604, 0.309552569975, -0.205539243633, -0.497043585027, 0.645622321029, 0.173007028285, -0.335039107286, 0.057325093568, -0.271921543048, 0.211985233143, 0.754720592187, 0.483804205078, -0.645991271674, -0.431623661140, 0.917464264471, 0.481820068657, 0.968187489149, 0.034619328690, 0.509609763385, -0.919387775095, 0.503276912408, -0.831363252242, 0.672486724694, -0.539306308255, -0.131801002154, -0.760998658513, 0.068148945241, 0.431135640962, 0.603761911866, 0.094939023607, -0.202716461984, -0.865823086598, -0.246461370843, 0.731326357993, -0.282282636542, 0.426825612756, 0.042613550851, -0.745187223256, 0.986234566961, -0.776290267733, -0.783273937001, 0.842605452334, 0.549561055702, 0.513268355062, 0.640955468311, 0.224752689092, 0.924868257906, 0.451338892544, -0.691978071880, -0.809809502385, 0.641994090044, 0.710503781834, -0.341602839866, 0.824254844198, -0.513481263424, 0.436272757059, 0.257891752223, 0.256222395868, 0.151214754920, -0.225748301791, -0.854399273866, -0.341300876024, 0.794130605885, 0.119739359466, -0.527082624111, 0.050621599094, 0.945639464269, 0.407736346989, 0.359276144500, 0.465822781998, 0.930298609121, -0.818747351040, 0.188613130355, 0.169150353456, -0.661555185591, -0.161898719292, -0.937868443401, 0.674718120863, 0.557085059762, -0.957101790449, 0.762346018775, -0.969290794044, 0.948966756638, -0.962415733484, -0.752546608429, -0.889791049765, 0.304112059707, 0.960164572677, -0.374735993776, -0.769977342364, 0.861642304012, 0.152145109456, 0.817654753552, 0.643508807945, -0.115234116665, 0.221046475438, -0.499654977678, 0.244260948970, -0.932560844393, 0.407409057234, 0.487058817445, 0.969593787923, -0.243069156201, -0.277626090603, -0.244541927947, 0.155441970391, -0.000319167253, -0.949532148169, -0.387100974077, 0.461774358585, 0.560285681454, 0.711119547086, 0.220163597903, 0.016659681397, 0.990354146661, 0.763312059070, 0.346708952586, -0.942956546101, 0.232858758216, -0.585050724444, -0.596559855309, -0.876422653890, 0.889146375158, 0.063588733480, 0.125864296364, -0.732470009600, -0.142256279752, -0.743757295986, -0.198626663680, 0.818436954843, 0.674680910292, -0.622598730962, 0.709995766988, 0.138498571566, 0.983196962357, 0.271553967100, -0.248790506750, -0.701730029655, 0.723723339410, 0.204668569928, -0.638799843135, -0.495223250676, 0.375130880342, 0.462218688501, -0.714779563882, -0.198077960197, -0.662022784312, -0.077641062748, -0.894494829636, 0.180808456545, 0.408763378165, -0.375348699793, -0.328482480801, 0.807563880490, -0.459478503397, 0.233516804917, 0.201855191109, -0.988446156060, 0.351580484398, -0.829445996388, -0.803605239177, 0.518802556468, -0.058217403374, 0.673081391708, 0.335456269607, 0.579509404864, 0.876431365003, 0.150974832424, -0.540504743215, -0.050282891661, -0.480839782151, -0.298963909155, 0.755040782637, -0.713143240635, -0.332610590428, -0.306932050550, 0.541665814218, 0.383357763106, -0.139180677723, -0.045674105016, 0.829492231989, -0.572099748071, 0.251326035081, 0.192358522433, -0.782033962729, 0.987247591925, -0.153571660629, -0.856699932663, -0.065641926965, -0.727319768709, -0.134945375129, -0.691940847422, -0.453750347592, 0.238651146843, -0.998807527370, 0.687963020475, 0.571254717916, 0.247651186774, 0.922843738833, 0.553777726483, 0.706435556126, -0.541550687250, -0.899983076325, -0.499777239198, 0.213711133056, -0.585480751412, -0.455636048139, -0.308826411531, 0.105076800820, -0.749992123357, -0.569654040837, 0.164771301618, 0.873520181875, 0.555360415703, -0.234989105180, -0.261106392041, -0.862349062026, 0.098437669757, 0.454214772050, -0.133298656590, 0.783920758797, 0.326292178099, 0.049707539608, 0.112037242429, -0.613437680403, 0.790602894874, 0.328373181832, -0.225023768478, -0.384334759503, 0.500102479285, 0.180053355510, -0.353624286045, 0.470020295810, -0.294160312666, -0.233888373461, -0.168316806351, 0.843115227492, 0.290675287400, 0.695850345033, 0.955778013424, -0.534907508626, 0.561269328360, 0.619170817972, -0.745524116530, -0.836964243080, 0.441031733522, -0.979231269250];
END_VAR

iI := iI + 1;
IF ((iI > 9999) OR (iI < 0)) THEN
	iI := 0;
END_IF

rY := arRauschen[iI]*rVerstaerkung;

(*
# Pyhtonskript zur Erzeugung der Zufallszahlen
import math
import random
##############################################################################   
def genoRauschen():
    # arRauschen: ARRAY [0..2] OF REAL := [0.0, 1.0, 2.0];
    lineOut = "arRauschen: ARRAY [0..9999] OF REAL := ["
    for i in range(10000):
        rndNr = random.random()*2 - 1.0
        print(rndNr)
        lineOut = lineOut + "{:.12f}".format(rndNr) + ", "
    lineOut = lineOut[:len(lineOut)-2] + "];\n"
    
    print(lineOut)

    fileName = "rauschen.txt"    
    fileRef = open(fileName, 'w')
    fileRef.write(lineOut)
    fileRef.close()
    
##############################################################################   
if __name__ == "__main__":
   genoRauschen()
*)

END_FUNCTION_BLOCK

// REGELUNGSTECHNIK/RealToInt
FUNCTION RealToInt : REAL
VAR_INPUT
	rIn: REAL;
END_VAR
VAR
END_VAR

RealToInt := TO_REAL(floor(rIn));

END_FUNCTION

// REGELUNGSTECHNIK/RealToUInt
FUNCTION RealToUInt : UINT
VAR_INPUT
	rIn: REAL;
END_VAR
VAR
END_VAR

RealToUInt := REAL_TO_UINT(rIn);

END_FUNCTION

// REGELUNGSTECHNIK/Regler
{attribute 'FBVisuCreator'}
{attribute 'FBVisuCreatorPrefix' :=  'RET_VISU_'}
FUNCTION_BLOCK PUBLIC Regler
VAR_INPUT
	{attribute 'FBVisuCreatorCustomName' := 'e'}
	{attribute 'FBVisuCreatorFormatString' := '%1.3f'}
	rE: REAL; // Regelfehler e
	{attribute 'FBVisuCreatorCustomName' := 'y_FF'}
	{attribute 'FBVisuCreatorFormatString' := '%1.3f'}
	rY_FF: REAL; // Vorsteuerung
	{attribute 'FBVisuCreatorCustomName' := 'Reglertyp'}
	{attribute 'FBVisuCreatorFormatString' := 'd'}
	eTyp:  eReglertyp;
	{attribute 'FBVisuCreatorBoolColor' := 'Red'}
	{attribute 'FBVisuCreatorCustomName' := 'Reset'}
	bReset: BOOL;
	{attribute 'FBVisuCreatorFormatString' := '%1.3f'}
	rKr: REAL; // Verstärkung Kr
	{attribute 'FBVisuCreatorFormatString' := '%1.3f'}
	rTn: REAL; // Nachstellzeit Tn
	{attribute 'FBVisuCreatorFormatString' := '%1.3f'}
	rTv: REAL; // Vorhaltezeit Tv
	{attribute 'FBVisuCreatorFormatString' := '%1.3f'}
	rTvz: REAL; // Zeitkonstante T1 für reales DT1-Verhalten
	{attribute 'FBVisuCreatorBoolColor' := 'Red'}
	bEnable_AWU: BOOL := TRUE;  // Aktivierung Anti-WindUp
	{attribute 'FBVisuCreatorFormatString' := '%1.3f'}
	rYlim_max: REAL; // Oberes Limit Anti-WindUp
	{attribute 'FBVisuCreatorFormatString' := '%1.3f'}
	rYlim_min: REAL; // Unteres Limit Anti-WindUp
END_VAR
VAR_OUTPUT
	{attribute 'FBVisuCreatorFormatString' := '%1.3f'}
	rY_RE: REAL;
	{attribute 'FBVisuCreatorFormatString' := '%1.3f'}
	rProportional: REAL;
	{attribute 'FBVisuCreatorFormatString' := '%1.3f'}
	rIntegral: REAL;
	{attribute 'FBVisuCreatorFormatString' := '%1.3f'}
	rDifferential: REAL;
	{attribute 'FBVisuCreatorBoolColor' := 'Red'}
	bAct_UL: BOOL := FALSE;
	{attribute 'FBVisuCreatorBoolColor' := 'Red'}
	bAct_LL: BOOL := FALSE;
END_VAR
VAR 
	dt1: DT1;	

	// Werden in Aktion eReglertyp gesetzt
	bEnKr: BOOL; // Freigabesignal P-Anteil
	bEnTn: BOOL; // Freigabesignal I-Anteil
	bEnTv: BOOL; // Freigabesignal D-Anteil
	//
	
	rIntegralCalc: REAL;
	
	rDy: REAL;
	rDx: REAL;
	rXeAlt: REAL;
	rYcalc: REAL;
	rYcalc_lim: REAL;
	
	rAvoidZero: REAL := 0.001;
	tonStartup: TON;
	bResetTvz: BOOL;
	bP_Regler: BOOL;
	bI_Regler: BOOL;
	bPI_Regler: BOOL;
	bPDT1_Regler: BOOL;
	bPIDT1_Regler: BOOL;
END_VAR

// Revisionhistory:
// -------------------------------------------------------------------------------------------------------------
// 2020-12-02, tr
// - Struktur/Implementation entspricht 1:1 derjenigen von BORIS mit Begrenzung Anti-WindUp Halt
// - Anti-WindUp komplett innerhalb dieses FB implementiert
// - zusätzliche Eingangsgrösse (rY_FF) für Einkopplung Vorsteuerungsanteil der Stellgrösse

// Grundlegende Reglerstruktur PID-T1-Regler:
// G(jw) = Kr*[1+1/(Tn*jw)+(Tv*jw/(1+Tvz*jw)]

Reglertyp();

///////////////////////////////////////////////////////////////////////////////////////////////////////////////
// Berechnung P-Anteil
IF bEnKr THEN // P-Anteil aktiv?
	rProportional := rKr*rE;
ELSE
	rKr := 1.0; // muss gesetzt werden, da sonst I-Anteil bei reinem I-Regler, aufgrund Struktur, nicht funktionieren würde.
	rProportional := 0;
END_IF

///////////////////////////////////////////////////////////////////////////////////////////////////////////////
// Berechnung I-Anteil
IF bEnTn THEN // I-Anteil aktiv?
	rIntegralCalc := rKr*(rE*RET_COMMON.rDt)/MAX(rTn,rAvoidZero);
ELSE
	rIntegral := 0;
END_IF

///////////////////////////////////////////////////////////////////////////////////////////////////////////////
// Auswertung Anti-WindUp, angepasst: 1.12.2020, tr
IF (rIntegral + rY_FF) >= (rYlim_max - rY_FF) AND rE > 0 AND bEnable_AWU THEN // I-Anteil halten, im Fall yI (nur I-Anteil) am oberen Limit und w > x
	rIntegral := rIntegral;
ELSIF (rIntegral + rY_FF) <= (rYlim_min + rY_FF) AND rE < 0 AND bEnable_AWU THEN // I-Anteil halten, im Fall yI (nur I-Anteil) am unteren Limit und w < x
	rIntegral := rIntegral;
ELSE
	rIntegral := rIntegral+ rIntegralCalc; // Integrieren / Summieren
END_IF

///////////////////////////////////////////////////////////////////////////////////////////////////////////////
// Berechnung DT1-Anteil, neu mittels Aufruf DT1-Grundglied realisiert
IF bEnTv AND (rTvz >= 2.0*RET_COMMON.rDt) THEN
	dt1(rE:=rKr*rE, rTv:=rTv , rTvz:=rTvz, rA=>rDifferential);
ELSE
	rDifferential := 0;
END_IF

///////////////////////////////////////////////////////////////////////////////////////////////////////////////
// Addition aller drei Teilkomponenten (P,I und DT1-Anteil)
// Die Implementation der Begrenzung (Anti-WindUp) entspricht der Umsetzung von BORIS, d.h. solange die Summe
// der beiden Anteile (P + I) ausserhalb der Limits sind wird das entsprechende Limit + D-Anteil als 
// Stellgrösse ausgegeben -> siehe nachfolgende Zeilen. Ansonsten werden sämtliche drei Anteile (P + I + D)
// addiert. Anpassung: 1.12.2020, tr
IF rProportional + rIntegral + rY_FF >= (rYlim_max - rY_FF) AND bEnable_AWU THEN
	rYcalc := rYlim_max + rDifferential;

ELSIF rProportional + rIntegral + rY_FF <= (rYlim_min + rY_FF) AND bEnable_AWU  THEN
	rYcalc := rYlim_min + rDifferential;

ELSE
	rYcalc := rProportional + rIntegral + rY_FF + rDifferential;
END_IF


///////////////////////////////////////////////////////////////////////////////////////////////////////////////
// Anti-WindUp
IF bEnable_AWU THEN
	IF rYcalc <= rYlim_max AND rYcalc >= rYlim_min THEN
		bAct_UL := FALSE;
		bAct_LL := FALSE;
	ELSIF rYcalc > rYlim_max THEN
			bAct_UL := TRUE;
			bAct_LL := FALSE;
	ELSIF rYcalc < rYlim_min THEN
		bAct_LL := TRUE;
		bAct_UL := FALSE;
	END_IF
	rY_RE := LIMIT(rYlim_min, rYcalc, rYlim_max);
ELSE
	rY_RE := rYcalc;
	bAct_LL := FALSE;
	bAct_UL := FALSE;
END_IF

IF bReset THEN
	this^.reset();
END_IF

ACTION Reglertyp:
// Auswahl möglicher Reglerkonfigurationen
CASE eTyp OF
	 eReglertyp.P:
	 	bP_Regler := TRUE;
		bI_Regler := FALSE;
		bPI_Regler := FALSE;
		bPDT1_Regler := FALSE;
		bPIDT1_Regler := FALSE;
		bEnKr := TRUE; // Freigabesignal P-Anteil
		bEnTn := FALSE; // Freigabesignal I-Anteil
		bEnTv := FALSE; // Freigabesignal D-Anteil;

	eReglertyp.I:
		bP_Regler := FALSE;
		bI_Regler := TRUE;
		bPI_Regler := FALSE;
		bPDT1_Regler := FALSE;
		bPIDT1_Regler := FALSE;
	 	bEnKr := FALSE; // Freigabesignal P-Anteil
		bEnTn := TRUE; // Freigabesignal I-Anteil
		bEnTv := FALSE; // Freigabesignal D-Anteil
		
		
	 eReglertyp.PI:
	 	bP_Regler := FALSE;
		bI_Regler := FALSE;
		bPI_Regler := TRUE;
		bPDT1_Regler := FALSE;
		bPIDT1_Regler := FALSE;
	 	bEnKr := TRUE; // Freigabesignal P-Anteil
		bEnTn := TRUE; // Freigabesignal I-Anteil
		bEnTv := FALSE; // Freigabesignal D-Anteil
				
	eReglertyp.PDT1:
		bP_Regler := FALSE;
		bI_Regler := FALSE;
		bPI_Regler := FALSE;
		bPDT1_Regler := TRUE;
		bPIDT1_Regler := FALSE;
	 	bEnKr := TRUE; // Freigabesignal P-Anteil
		bEnTn := FALSE; // Freigabesignal I-Anteil
		bEnTv := TRUE; // Freigabesignal D-Anteil
		
	eReglertyp.PIDT1:
		bP_Regler := FALSE;
		bI_Regler := FALSE;
		bPI_Regler := FALSE;
		bPDT1_Regler := FALSE;
		bPIDT1_Regler := TRUE;
	 	bEnKr := TRUE; // Freigabesignal P-Anteil
		bEnTn := TRUE; // Freigabesignal I-Anteil
		bEnTv := TRUE; // Freigabesignal D-Anteil
	
END_CASE
END_ACTION

ACTION reset:
rProportional := 0.0;
rIntegral := 0.0;
rDifferential := 0.0;
dt1.reset();
rY_RE := 0.0;
//rTv := 0.0;
rY_RE := 0.0;
END_ACTION

END_FUNCTION_BLOCK

// REGELUNGSTECHNIK/Signalgenerator
{attribute 'FBVisuCreator'}
{attribute 'FBVisuCreatorPrefix' :=  'RET_VISU_'}
FUNCTION_BLOCK Signalgenerator
VAR_INPUT
	{attribute 'FBVisuCreatorCustomName' := 'Typ'}
	{attribute 'FBVisuCreatorFormatString' := 'd'}
	eTyp: eSignalform := eSignalform.OFF;
	{attribute 'FBVisuCreatorCustomName' := 'Offset'}
	{attribute 'FBVisuCreatorFormatString' := '%1.3f'}
	rOffset: REAL := 0.0;
	{attribute 'FBVisuCreatorCustomName' := 'Offset_Rampe'}
	{attribute 'FBVisuCreatorFormatString' := '%1.3f'}
	rRampe: REAL := 0.0;
	{attribute 'FBVisuCreatorCustomName' := 'Rampensteilheit'}
	{attribute 'FBVisuCreatorFormatString' := '%1.3f'}
	rdW_dt: REAL := 1.0; // entspricht Steilheit der Rampe, d.h. 1.0 --> 1.0 dW/dt
	{attribute 'FBVisuCreatorCustomName' := 'Amplitude'}
	{attribute 'FBVisuCreatorFormatString' := '%1.3f'}
	rAmplitude: REAL := 1.0;
	{attribute 'FBVisuCreatorCustomName' := 'Frequenz [Hz]'}
	{attribute 'FBVisuCreatorFormatString' := '%1.5f'}
	rFrequenz: REAL := 1.0;
	{attribute 'FBVisuCreatorCustomName' := 'Phasenverschiebung [°]'}
	{attribute 'FBVisuCreatorFormatString' := '%1.1f'}
	rPhi: REAL := 0.0;
	{attribute 'FBVisuCreatorBoolColor' := 'Red'}
	bRauschen: BOOL;
	{attribute 'FBVisuCreatorFormatString' := '%1.3f'}
	rRauschenVerstaerkung: REAL;
END_VAR
VAR_OUTPUT
	{attribute 'FBVisuCreatorFormatString' := '%1.3f'}
	rY: REAL;
END_VAR
VAR
	rZeit: REAL;
	rSumme: REAL;
	rauschen: Rauschen := (rVerstaerkung := 1.0);
	rYsin: REAL;
	rYasin: REAL;
END_VAR
VAR CONSTANT
	rPi: REAL := 3.141592653589790;
END_VAR

rZeit := rZeit + RET_COMMON.rDt;

CASE eTyp OF
	eSignalform.OFF:
		rY := 0.0;
		rSumme := 0.0;
	
	eSignalform.OFFSET:
		rY := rOffset;
		rRampe := rOffset;
		
	eSignalform.RAMPE:
		IF rY < rRampe THEN
			rSumme := rSumme + rdW_dt*RET_COMMON.rDt;
		ELSIF rY > rRampe THEN
			rSumme := rSumme - rdW_dt*RET_COMMON.rDt;
		ELSE
			rY := rRampe;
		END_IF
		
		IF rY = rRampe THEN// AntiWindUp
			rY := rRampe;
			rOffset := rRampe; // neuer Startpunkt für Rampe setzen
		ELSE
			rY := rOffset + rSumme;
		END_IF
			
	eSignalform.RECHTECK:
		rY := SIN(2*rPi*rFrequenz*rZeit + rPhi*rPi/180.0);
		IF rY >= 0.0 THEN
			rY := rAmplitude;
		ELSIF rY < 0.0 THEN
			rY :=  -rAmplitude;
		END_IF
		rY := LIMIT(-500.0, rY + rOffset, 500.0);
		rRampe := rOffset;

	eSignalform.DREIECK:
		rYsin := SIN(2*rPi*rFrequenz*rZeit + rPhi*rPi/180.0);
		rYasin := 2*ASIN(rYsin)/rPi;
		rY := rAmplitude*rYasin + rOffset;
		
	eSignalform.SINUS:
		rY := rAmplitude*SIN(2*rPi*rFrequenz*rZeit + rPhi*rPi/180.0) + rOffset;
		rRampe := rOffset;
		
	ELSE
		eTyp := eSignalform.OFF;
END_CASE
IF bRauschen AND (eTyp <> eSignalform.OFF) THEN
	rauschen(rVerstaerkung := rRauschenVerstaerkung);
	rY := rY + rauschen.rY;
END_IF

END_FUNCTION_BLOCK

// /RET_VISU_Signalgenerator
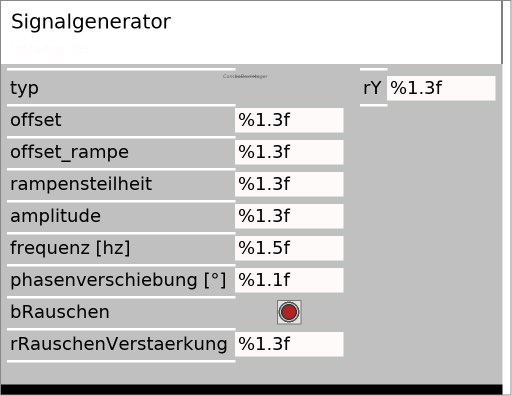
VISUALIZATION RET_VISU_Signalgenerator  // 512x396
VAR_INPUT
   {attribute 'parameterstringof' := 'm_Input_FB'}
   m_Input_INST_Str : STRING;
END_VAR
VAR_IN_OUT
   m_Input_FB : Signalgenerator;
END_VAR
    RoundedRectangle (0,0 502x81)
    RoundedRectangle (0,354 502x40)
    Rectangle (0,64 502x320)
    PushSwitch (277,300 24x24), variable: m_Input_FB.bRauschen, behaviour: TOGGLE, style: Switch-PushSwitch-Red
    Rectangle (8,8 502x27), "Signalgenerator"
    Rectangle (8,35 502x27), "Instance: %s", text variable: m_Input_INST_Str
    Rectangle (7,68 228x2)
    Rectangle (7,76 228x24), "typ"
    Rectangle (7,104 228x2)
    Rectangle (235,108 108x24), "%1.3f", text variable: m_Input_FB.rOffset
        OnMouseClick: write the text variable via Default
    Rectangle (7,108 228x24), "offset"
    Rectangle (7,136 228x2)
    Rectangle (235,140 108x24), "%1.3f", text variable: m_Input_FB.rRampe
        OnMouseClick: write the text variable via Default
    Rectangle (7,140 228x24), "offset_rampe"
    Rectangle (7,168 228x2)
    Rectangle (235,172 108x24), "%1.3f", text variable: m_Input_FB.rdW_dt
        OnMouseClick: write the text variable via Default
    Rectangle (7,172 228x24), "rampensteilheit"
    Rectangle (7,200 228x2)
    Rectangle (235,204 108x24), "%1.3f", text variable: m_Input_FB.rAmplitude
        OnMouseClick: write the text variable via Default
    Rectangle (7,204 228x24), "amplitude"
    Rectangle (7,232 228x2)
    Rectangle (235,236 108x24), "%1.5f", text variable: m_Input_FB.rFrequenz
        OnMouseClick: write the text variable via Default
    Rectangle (7,236 228x24), "frequenz [hz]"
    Rectangle (7,264 228x2)
    Rectangle (235,268 108x24), "%1.1f", text variable: m_Input_FB.rPhi
        OnMouseClick: write the text variable via Default
    Rectangle (7,268 228x24), "phasenverschiebung [°]"
    Rectangle (7,296 228x2)
    Rectangle (7,300 228x24), "bRauschen"
    Rectangle (7,328 228x2)
    Rectangle (235,332 108x24), "%1.3f", text variable: m_Input_FB.rRauschenVerstaerkung
        OnMouseClick: write the text variable via Default
    Rectangle (7,332 228x24), "rRauschenVerstaerkung"
    Rectangle (7,360 228x2)
    Rectangle (360,68 27x2)
    Rectangle (387,76 108x24), "%1.3f", text variable: m_Input_FB.rY
    Rectangle (360,76 27x24), "rY"
    Rectangle (360,104 27x2)
    Frame (235,76 108x24), input disabled if: False
        shows VISU_HELPER_Combobox_eSignalform(varEnum := m_Input_FB.eTyp)
END_VISUALIZATION

// /RET_VISU_Regler
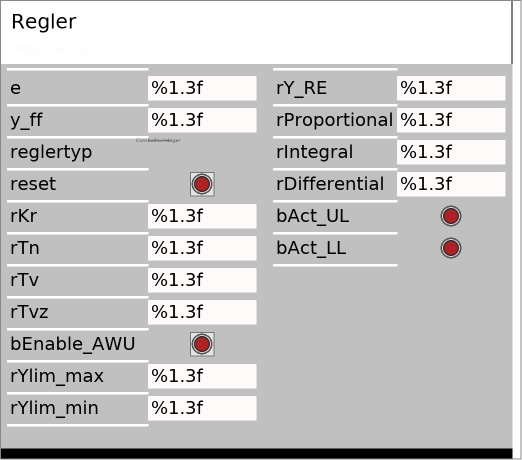
VISUALIZATION RET_VISU_Regler  // 522x460
VAR_INPUT
   {attribute 'parameterstringof' := 'm_Input_FB'}
   m_Input_INST_Str : STRING;
END_VAR
VAR_IN_OUT
   m_Input_FB : Regler;
END_VAR
    RoundedRectangle (0,0 512x81)
    RoundedRectangle (0,418 512x40)
    Rectangle (0,64 512x384)
    Lamp1 (439,204 24x24), variable: m_Input_FB.bAct_UL, style: Lamp-Lamp1-Red
    Lamp1 (439,236 24x24), variable: m_Input_FB.bAct_LL, style: Lamp-Lamp1-Red
    PushSwitch (190,172 24x24), variable: m_Input_FB.bReset, behaviour: TOGGLE, style: Switch-PushSwitch-Red
    PushSwitch (190,332 24x24), variable: m_Input_FB.bEnable_AWU, behaviour: TOGGLE, style: Switch-PushSwitch-Red
    Rectangle (8,8 512x27), "Regler"
    Rectangle (8,35 512x27), "Instance: %s", text variable: m_Input_INST_Str
    Rectangle (7,68 141x2)
    Rectangle (148,76 108x24), "%1.3f", text variable: m_Input_FB.rE
        OnMouseClick: write the text variable via Default
    Rectangle (7,76 141x24), "e"
    Rectangle (7,104 141x2)
    Rectangle (148,108 108x24), "%1.3f", text variable: m_Input_FB.rY_FF
        OnMouseClick: write the text variable via Default
    Rectangle (7,108 141x24), "y_ff"
    Rectangle (7,136 141x2)
    Rectangle (7,140 141x24), "reglertyp"
    Rectangle (7,168 141x2)
    Rectangle (7,172 141x24), "reset"
    Rectangle (7,200 141x2)
    Rectangle (148,204 108x24), "%1.3f", text variable: m_Input_FB.rKr
        OnMouseClick: write the text variable via Default
    Rectangle (7,204 141x24), "rKr"
    Rectangle (7,232 141x2)
    Rectangle (148,236 108x24), "%1.3f", text variable: m_Input_FB.rTn
        OnMouseClick: write the text variable via Default
    Rectangle (7,236 141x24), "rTn"
    Rectangle (7,264 141x2)
    Rectangle (148,268 108x24), "%1.3f", text variable: m_Input_FB.rTv
        OnMouseClick: write the text variable via Default
    Rectangle (7,268 141x24), "rTv"
    Rectangle (7,296 141x2)
    Rectangle (148,300 108x24), "%1.3f", text variable: m_Input_FB.rTvz
        OnMouseClick: write the text variable via Default
    Rectangle (7,300 141x24), "rTvz"
    Rectangle (7,328 141x2)
    Rectangle (7,332 141x24), "bEnable_AWU"
    Rectangle (7,360 141x2)
    Rectangle (148,364 108x24), "%1.3f", text variable: m_Input_FB.rYlim_max
        OnMouseClick: write the text variable via Default
    Rectangle (7,364 141x24), "rYlim_max"
    Rectangle (7,392 141x2)
    Rectangle (148,396 108x24), "%1.3f", text variable: m_Input_FB.rYlim_min
        OnMouseClick: write the text variable via Default
    Rectangle (7,396 141x24), "rYlim_min"
    Rectangle (7,424 141x2)
    Rectangle (273,68 124x2)
    Rectangle (397,76 108x24), "%1.3f", text variable: m_Input_FB.rY_RE
    Rectangle (273,76 124x24), "rY_RE"
    Rectangle (273,104 124x2)
    Rectangle (397,108 108x24), "%1.3f", text variable: m_Input_FB.rProportional
    Rectangle (273,108 124x24), "rProportional"
    Rectangle (273,136 124x2)
    Rectangle (397,140 108x24), "%1.3f", text variable: m_Input_FB.rIntegral
    Rectangle (273,140 124x24), "rIntegral"
    Rectangle (273,168 124x2)
    Rectangle (397,172 108x24), "%1.3f", text variable: m_Input_FB.rDifferential
    Rectangle (273,172 124x24), "rDifferential"
    Rectangle (273,200 124x2)
    Rectangle (273,204 124x24), "bAct_UL"
    Rectangle (273,232 124x2)
    Rectangle (273,236 124x24), "bAct_LL"
    Rectangle (273,264 124x2)
    Frame (148,140 108x24), input disabled if: False
        shows VISU_HELPER_Combobox_eReglertyp(varEnum := m_Input_FB.eTyp)
END_VISUALIZATION

// /RET_VISU_Totband
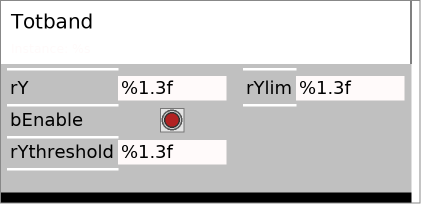
VISUALIZATION RET_VISU_Totband  // 421x204
VAR_INPUT
   {attribute 'parameterstringof' := 'm_Input_FB'}
   m_Input_INST_Str : STRING;
END_VAR
VAR_IN_OUT
   m_Input_FB : Totband;
END_VAR
    RoundedRectangle (0,0 411x81)
    RoundedRectangle (0,162 411x40)
    Rectangle (0,64 411x128)
    PushSwitch (160,108 24x24), variable: m_Input_FB.bEnable, behaviour: TOGGLE, style: Switch-PushSwitch-Red
    Rectangle (8,8 411x27), "Totband"
    Rectangle (8,35 411x27), "Instance: %s", text variable: m_Input_INST_Str
    Rectangle (7,68 111x2)
    Rectangle (118,76 108x24), "%1.3f", text variable: m_Input_FB.rY
        OnMouseClick: write the text variable via Default
    Rectangle (7,76 111x24), "rY"
    Rectangle (7,104 111x2)
    Rectangle (7,108 111x24), "bEnable"
    Rectangle (7,136 111x2)
    Rectangle (118,140 108x24), "%1.3f", text variable: m_Input_FB.rYthreshold
        OnMouseClick: write the text variable via Default
    Rectangle (7,140 111x24), "rYthreshold"
    Rectangle (7,168 111x2)
    Rectangle (243,68 53x2)
    Rectangle (296,76 108x24), "%1.3f", text variable: m_Input_FB.rYlim
    Rectangle (243,76 53x24), "rYlim"
    Rectangle (243,104 53x2)
END_VISUALIZATION

// /RET_VISU_Rauschen
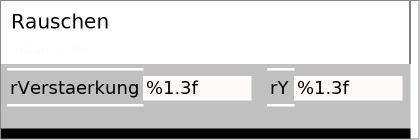
VISUALIZATION RET_VISU_Rauschen  // 420x140
VAR_INPUT
   {attribute 'parameterstringof' := 'm_Input_FB'}
   m_Input_INST_Str : STRING;
END_VAR
VAR_IN_OUT
   m_Input_FB : Rauschen;
END_VAR
    RoundedRectangle (0,0 410x81)
    RoundedRectangle (0,98 410x40)
    Rectangle (0,64 410x64)
    Rectangle (8,8 410x27), "Rauschen"
    Rectangle (8,35 410x27), "Instance: %s", text variable: m_Input_INST_Str
    Rectangle (7,68 136x2)
    Rectangle (143,76 108x24), "%1.3f", text variable: m_Input_FB.rVerstaerkung
        OnMouseClick: write the text variable via Default
    Rectangle (7,76 136x24), "rVerstaerkung"
    Rectangle (7,104 136x2)
    Rectangle (267,68 27x2)
    Rectangle (294,76 108x24), "%1.3f", text variable: m_Input_FB.rY
    Rectangle (267,76 27x24), "rY"
    Rectangle (267,104 27x2)
END_VISUALIZATION

// /RET_VISU_PTt
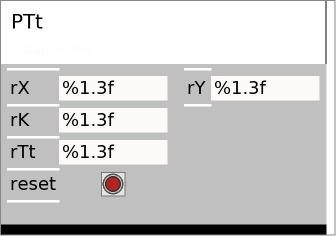
VISUALIZATION RET_VISU_PTt  // 336x236
VAR_INPUT
   {attribute 'parameterstringof' := 'm_Input_FB'}
   m_Input_INST_Str : STRING;
END_VAR
VAR_IN_OUT
   m_Input_FB : PTt;
END_VAR
    RoundedRectangle (0,0 326x81)
    RoundedRectangle (0,194 326x40)
    Rectangle (0,64 326x160)
    PushSwitch (101,172 24x24), variable: m_Input_FB.bReset, behaviour: TOGGLE, style: Switch-PushSwitch-Red
    Rectangle (8,8 326x27), "PTt"
    Rectangle (8,35 326x27), "Instance: %s", text variable: m_Input_INST_Str
    Rectangle (7,68 52x2)
    Rectangle (59,76 108x24), "%1.3f", text variable: m_Input_FB.rX
        OnMouseClick: write the text variable via Default
    Rectangle (7,76 52x24), "rX"
    Rectangle (7,104 52x2)
    Rectangle (59,108 108x24), "%1.3f", text variable: m_Input_FB.rK
        OnMouseClick: write the text variable via Default
    Rectangle (7,108 52x24), "rK"
    Rectangle (7,136 52x2)
    Rectangle (59,140 108x24), "%1.3f", text variable: m_Input_FB.rTt
        OnMouseClick: write the text variable via Default
    Rectangle (7,140 52x24), "rTt"
    Rectangle (7,168 52x2)
    Rectangle (7,172 52x24), "reset"
    Rectangle (7,200 52x2)
    Rectangle (184,68 27x2)
    Rectangle (211,76 108x24), "%1.3f", text variable: m_Input_FB.rY
    Rectangle (184,76 27x24), "rY"
    Rectangle (184,104 27x2)
END_VISUALIZATION

// /RET_VISU_PT2s
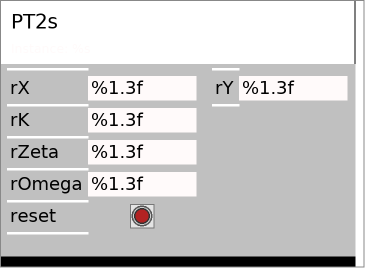
VISUALIZATION RET_VISU_PT2s  // 365x268
VAR_INPUT
   {attribute 'parameterstringof' := 'm_Input_FB'}
   m_Input_INST_Str : STRING;
END_VAR
VAR_IN_OUT
   m_Input_FB : PT2s;
END_VAR
    RoundedRectangle (0,0 355x81)
    RoundedRectangle (0,226 355x40)
    Rectangle (0,64 355x192)
    PushSwitch (130,204 24x24), variable: m_Input_FB.bReset, behaviour: TOGGLE, style: Switch-PushSwitch-Red
    Rectangle (8,8 355x27), "PT2s"
    Rectangle (8,35 355x27), "Instance: %s", text variable: m_Input_INST_Str
    Rectangle (7,68 81x2)
    Rectangle (88,76 108x24), "%1.3f", text variable: m_Input_FB.rX
        OnMouseClick: write the text variable via Default
    Rectangle (7,76 81x24), "rX"
    Rectangle (7,104 81x2)
    Rectangle (88,108 108x24), "%1.3f", text variable: m_Input_FB.rK
        OnMouseClick: write the text variable via Default
    Rectangle (7,108 81x24), "rK"
    Rectangle (7,136 81x2)
    Rectangle (88,140 108x24), "%1.3f", text variable: m_Input_FB.rZeta
        OnMouseClick: write the text variable via Default
    Rectangle (7,140 81x24), "rZeta"
    Rectangle (7,168 81x2)
    Rectangle (88,172 108x24), "%1.3f", text variable: m_Input_FB.rOmega
        OnMouseClick: write the text variable via Default
    Rectangle (7,172 81x24), "rOmega"
    Rectangle (7,200 81x2)
    Rectangle (7,204 81x24), "reset"
    Rectangle (7,232 81x2)
    Rectangle (212,68 27x2)
    Rectangle (239,76 108x24), "%1.3f", text variable: m_Input_FB.rY
    Rectangle (212,76 27x24), "rY"
    Rectangle (212,104 27x2)
END_VISUALIZATION

// /RET_VISU_PT2
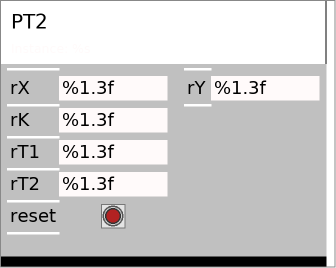
VISUALIZATION RET_VISU_PT2  // 336x268
VAR_INPUT
   {attribute 'parameterstringof' := 'm_Input_FB'}
   m_Input_INST_Str : STRING;
END_VAR
VAR_IN_OUT
   m_Input_FB : PT2;
END_VAR
    RoundedRectangle (0,0 326x81)
    RoundedRectangle (0,226 326x40)
    Rectangle (0,64 326x192)
    PushSwitch (101,204 24x24), variable: m_Input_FB.bReset, behaviour: TOGGLE, style: Switch-PushSwitch-Red
    Rectangle (8,8 326x27), "PT2"
    Rectangle (8,35 326x27), "Instance: %s", text variable: m_Input_INST_Str
    Rectangle (7,68 52x2)
    Rectangle (59,76 108x24), "%1.3f", text variable: m_Input_FB.rX
        OnMouseClick: write the text variable via Default
    Rectangle (7,76 52x24), "rX"
    Rectangle (7,104 52x2)
    Rectangle (59,108 108x24), "%1.3f", text variable: m_Input_FB.rK
        OnMouseClick: write the text variable via Default
    Rectangle (7,108 52x24), "rK"
    Rectangle (7,136 52x2)
    Rectangle (59,140 108x24), "%1.3f", text variable: m_Input_FB.rT1
        OnMouseClick: write the text variable via Default
    Rectangle (7,140 52x24), "rT1"
    Rectangle (7,168 52x2)
    Rectangle (59,172 108x24), "%1.3f", text variable: m_Input_FB.rT2
        OnMouseClick: write the text variable via Default
    Rectangle (7,172 52x24), "rT2"
    Rectangle (7,200 52x2)
    Rectangle (7,204 52x24), "reset"
    Rectangle (7,232 52x2)
    Rectangle (184,68 27x2)
    Rectangle (211,76 108x24), "%1.3f", text variable: m_Input_FB.rY
    Rectangle (184,76 27x24), "rY"
    Rectangle (184,104 27x2)
END_VISUALIZATION

// /RET_VISU_PT1
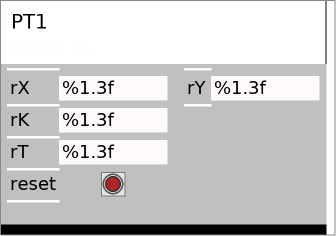
VISUALIZATION RET_VISU_PT1  // 336x236
VAR_INPUT
   {attribute 'parameterstringof' := 'm_Input_FB'}
   m_Input_INST_Str : STRING;
END_VAR
VAR_IN_OUT
   m_Input_FB : PT1;
END_VAR
    RoundedRectangle (0,0 326x81)
    RoundedRectangle (0,194 326x40)
    Rectangle (0,64 326x160)
    PushSwitch (101,172 24x24), variable: m_Input_FB.bReset, behaviour: TOGGLE, style: Switch-PushSwitch-Red
    Rectangle (8,8 326x27), "PT1"
    Rectangle (8,35 326x27), "Instance: %s", text variable: m_Input_INST_Str
    Rectangle (7,68 52x2)
    Rectangle (59,76 108x24), "%1.3f", text variable: m_Input_FB.rX
        OnMouseClick: write the text variable via Default
    Rectangle (7,76 52x24), "rX"
    Rectangle (7,104 52x2)
    Rectangle (59,108 108x24), "%1.3f", text variable: m_Input_FB.rK
        OnMouseClick: write the text variable via Default
    Rectangle (7,108 52x24), "rK"
    Rectangle (7,136 52x2)
    Rectangle (59,140 108x24), "%1.3f", text variable: m_Input_FB.rT
        OnMouseClick: write the text variable via Default
    Rectangle (7,140 52x24), "rT"
    Rectangle (7,168 52x2)
    Rectangle (7,172 52x24), "reset"
    Rectangle (7,200 52x2)
    Rectangle (184,68 27x2)
    Rectangle (211,76 108x24), "%1.3f", text variable: m_Input_FB.rY
    Rectangle (184,76 27x24), "rY"
    Rectangle (184,104 27x2)
END_VISUALIZATION

// /RET_VISU_P
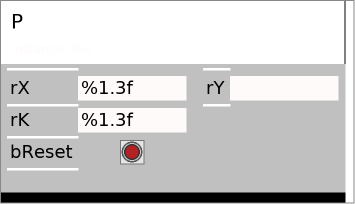
VISUALIZATION RET_VISU_P  // 355x204
VAR_INPUT
   {attribute 'parameterstringof' := 'm_Input_FB'}
   m_Input_INST_Str : STRING;
END_VAR
VAR_IN_OUT
   m_Input_FB : P;
END_VAR
    RoundedRectangle (0,0 345x81)
    RoundedRectangle (0,162 345x40)
    Rectangle (0,64 345x128)
    PushSwitch (120,140 24x24), variable: m_Input_FB.bReset, behaviour: TOGGLE, style: Switch-PushSwitch-Red
    Rectangle (8,8 345x27), "P"
    Rectangle (8,35 345x27), "Instance: %s", text variable: m_Input_INST_Str
    Rectangle (7,68 71x2)
    Rectangle (78,76 108x24), "%1.3f", text variable: m_Input_FB.rX
        OnMouseClick: write the text variable via Default
    Rectangle (7,76 71x24), "rX"
    Rectangle (7,104 71x2)
    Rectangle (78,108 108x24), "%1.3f", text variable: m_Input_FB.rK
        OnMouseClick: write the text variable via Default
    Rectangle (7,108 71x24), "rK"
    Rectangle (7,136 71x2)
    Rectangle (7,140 71x24), "bReset"
    Rectangle (7,168 71x2)
    Rectangle (203,68 27x2)
    Rectangle (230,76 108x24), text variable: m_Input_FB.rY
    Rectangle (203,76 27x24), "rY"
    Rectangle (203,104 27x2)
END_VISUALIZATION

// /RET_VISU_Limitierung
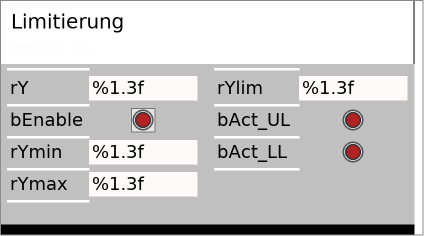
VISUALIZATION RET_VISU_Limitierung  // 424x236
VAR_INPUT
   {attribute 'parameterstringof' := 'm_Input_FB'}
   m_Input_INST_Str : STRING;
END_VAR
VAR_IN_OUT
   m_Input_FB : Limitierung;
END_VAR
    RoundedRectangle (0,0 414x81)
    RoundedRectangle (0,194 414x40)
    Rectangle (0,64 414x160)
    Lamp1 (341,108 24x24), variable: m_Input_FB.bAct_UL, style: Lamp-Lamp1-Red
    Lamp1 (341,140 24x24), variable: m_Input_FB.bAct_LL, style: Lamp-Lamp1-Red
    PushSwitch (131,108 24x24), variable: m_Input_FB.bEnable, behaviour: TOGGLE, style: Switch-PushSwitch-Red
    Rectangle (8,8 414x27), "Limitierung"
    Rectangle (8,35 414x27), "Instance: %s", text variable: m_Input_INST_Str
    Rectangle (7,68 82x2)
    Rectangle (89,76 108x24), "%1.3f", text variable: m_Input_FB.rY
        OnMouseClick: write the text variable via Default
    Rectangle (7,76 82x24), "rY"
    Rectangle (7,104 82x2)
    Rectangle (7,108 82x24), "bEnable"
    Rectangle (7,136 82x2)
    Rectangle (89,140 108x24), "%1.3f", text variable: m_Input_FB.rYmin
        OnMouseClick: write the text variable via Default
    Rectangle (7,140 82x24), "rYmin"
    Rectangle (7,168 82x2)
    Rectangle (89,172 108x24), "%1.3f", text variable: m_Input_FB.rYmax
        OnMouseClick: write the text variable via Default
    Rectangle (7,172 82x24), "rYmax"
    Rectangle (7,200 82x2)
    Rectangle (214,68 85x2)
    Rectangle (299,76 108x24), "%1.3f", text variable: m_Input_FB.rYlim
    Rectangle (214,76 85x24), "rYlim"
    Rectangle (214,104 85x2)
    Rectangle (214,108 85x24), "bAct_UL"
    Rectangle (214,136 85x2)
    Rectangle (214,140 85x24), "bAct_LL"
    Rectangle (214,168 85x2)
END_VISUALIZATION

// /RET_VISU_Kennlinie
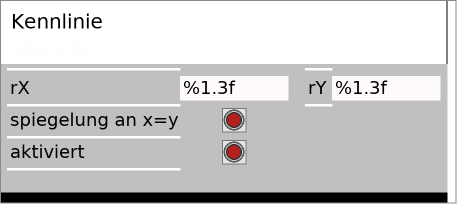
VISUALIZATION RET_VISU_Kennlinie  // 457x204
VAR_INPUT
   {attribute 'parameterstringof' := 'm_Input_FB'}
   m_Input_INST_Str : STRING;
END_VAR
VAR_IN_OUT
   m_Input_FB : Kennlinie;
END_VAR
    RoundedRectangle (0,0 447x81)
    RoundedRectangle (0,162 447x40)
    Rectangle (0,64 447x128)
    PushSwitch (222,108 24x24), variable: m_Input_FB.bSpiegelungXgY, behaviour: TOGGLE, style: Switch-PushSwitch-Red
    PushSwitch (222,140 24x24), variable: m_Input_FB.bAktiviert, behaviour: TOGGLE, style: Switch-PushSwitch-Red
    Rectangle (8,8 447x27), "Kennlinie"
    Rectangle (8,35 447x27), "Instance: %s", text variable: m_Input_INST_Str
    Rectangle (7,68 173x2)
    Rectangle (180,76 108x24), "%1.3f", text variable: m_Input_FB.rX
        OnMouseClick: write the text variable via Default
    Rectangle (7,76 173x24), "rX"
    Rectangle (7,104 173x2)
    Rectangle (7,108 173x24), "spiegelung an x=y"
    Rectangle (7,136 173x2)
    Rectangle (7,140 173x24), "aktiviert"
    Rectangle (7,168 173x2)
    Rectangle (305,68 27x2)
    Rectangle (332,76 108x24), "%1.3f", text variable: m_Input_FB.rY
    Rectangle (305,76 27x24), "rY"
    Rectangle (305,104 27x2)
END_VISUALIZATION

// /RET_VISU_Integrator
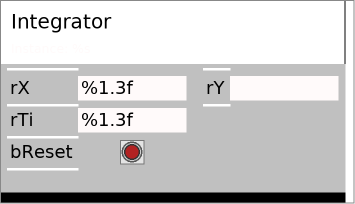
VISUALIZATION RET_VISU_Integrator  // 355x204
VAR_INPUT
   {attribute 'parameterstringof' := 'm_Input_FB'}
   m_Input_INST_Str : STRING;
END_VAR
VAR_IN_OUT
   m_Input_FB : Integrator;
END_VAR
    RoundedRectangle (0,0 345x81)
    RoundedRectangle (0,162 345x40)
    Rectangle (0,64 345x128)
    PushSwitch (120,140 24x24), variable: m_Input_FB.bReset, behaviour: TOGGLE, style: Switch-PushSwitch-Red
    Rectangle (8,8 345x27), "Integrator"
    Rectangle (8,35 345x27), "Instance: %s", text variable: m_Input_INST_Str
    Rectangle (7,68 71x2)
    Rectangle (78,76 108x24), "%1.3f", text variable: m_Input_FB.rX
        OnMouseClick: write the text variable via Default
    Rectangle (7,76 71x24), "rX"
    Rectangle (7,104 71x2)
    Rectangle (78,108 108x24), "%1.3f", text variable: m_Input_FB.rTi
        OnMouseClick: write the text variable via Default
    Rectangle (7,108 71x24), "rTi"
    Rectangle (7,136 71x2)
    Rectangle (7,140 71x24), "bReset"
    Rectangle (7,168 71x2)
    Rectangle (203,68 27x2)
    Rectangle (230,76 108x24), text variable: m_Input_FB.rY
    Rectangle (203,76 27x24), "rY"
    Rectangle (203,104 27x2)
END_VISUALIZATION

// /RET_VISU_DT1
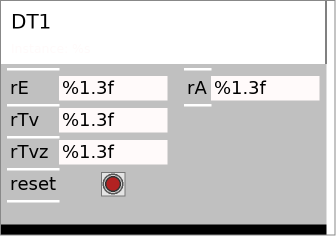
VISUALIZATION RET_VISU_DT1  // 336x236
VAR_INPUT
   {attribute 'parameterstringof' := 'm_Input_FB'}
   m_Input_INST_Str : STRING;
END_VAR
VAR_IN_OUT
   m_Input_FB : DT1;
END_VAR
    RoundedRectangle (0,0 326x81)
    RoundedRectangle (0,194 326x40)
    Rectangle (0,64 326x160)
    PushSwitch (101,172 24x24), variable: m_Input_FB.bReset, behaviour: TOGGLE, style: Switch-PushSwitch-Red
    Rectangle (8,8 326x27), "DT1"
    Rectangle (8,35 326x27), "Instance: %s", text variable: m_Input_INST_Str
    Rectangle (7,68 52x2)
    Rectangle (59,76 108x24), "%1.3f", text variable: m_Input_FB.rE
        OnMouseClick: write the text variable via Default
    Rectangle (7,76 52x24), "rE"
    Rectangle (7,104 52x2)
    Rectangle (59,108 108x24), "%1.3f", text variable: m_Input_FB.rTv
        OnMouseClick: write the text variable via Default
    Rectangle (7,108 52x24), "rTv"
    Rectangle (7,136 52x2)
    Rectangle (59,140 108x24), "%1.3f", text variable: m_Input_FB.rTvz
        OnMouseClick: write the text variable via Default
    Rectangle (7,140 52x24), "rTvz"
    Rectangle (7,168 52x2)
    Rectangle (7,172 52x24), "reset"
    Rectangle (7,200 52x2)
    Rectangle (184,68 27x2)
    Rectangle (211,76 108x24), "%1.3f", text variable: m_Input_FB.rA
    Rectangle (184,76 27x24), "rA"
    Rectangle (184,104 27x2)
END_VISUALIZATION

// /RET_VISU_KalmanFilter
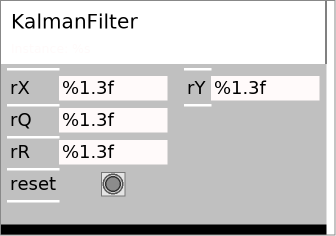
VISUALIZATION RET_VISU_KalmanFilter  // 336x236
VAR_INPUT
   {attribute 'parameterstringof' := 'm_Input_FB'}
   m_Input_INST_Str : STRING;
END_VAR
VAR_IN_OUT
   m_Input_FB : KalmanFilter;
END_VAR
    RoundedRectangle (0,0 326x81)
    RoundedRectangle (0,194 326x40)
    Rectangle (0,64 326x160)
    PushSwitch (101,172 24x24), variable: m_Input_FB.bReset, behaviour: TOGGLE, style: Switch-PushSwitch-Gray
    Rectangle (8,8 326x27), "KalmanFilter"
    Rectangle (8,35 326x27), "Instance: %s", text variable: m_Input_INST_Str
    Rectangle (7,68 52x2)
    Rectangle (59,76 108x24), "%1.3f", text variable: m_Input_FB.rX
        OnMouseClick: write the text variable via Default
    Rectangle (7,76 52x24), "rX"
    Rectangle (7,104 52x2)
    Rectangle (59,108 108x24), "%1.3f", text variable: m_Input_FB.rQ
        OnMouseClick: write the text variable via Default
    Rectangle (7,108 52x24), "rQ"
    Rectangle (7,136 52x2)
    Rectangle (59,140 108x24), "%1.3f", text variable: m_Input_FB.rR
        OnMouseClick: write the text variable via Default
    Rectangle (7,140 52x24), "rR"
    Rectangle (7,168 52x2)
    Rectangle (7,172 52x24), "reset"
    Rectangle (7,200 52x2)
    Rectangle (184,68 27x2)
    Rectangle (211,76 108x24), "%1.3f", text variable: m_Input_FB.rY
    Rectangle (184,76 27x24), "rY"
    Rectangle (184,104 27x2)
END_VISUALIZATION

// /VISU_HELPER_Combobox_eReglertyp
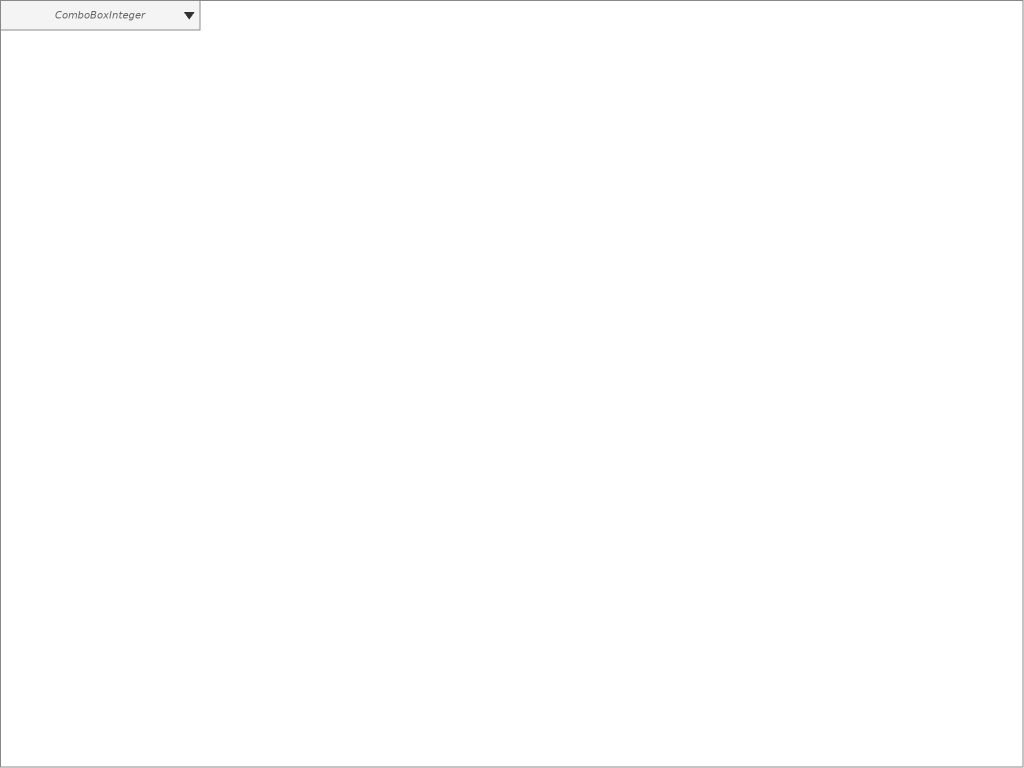
VISUALIZATION VISU_HELPER_Combobox_eReglertyp  // 1024x768
VAR_IN_OUT
    varEnum : eReglertyp;
END_VAR
    ComboBoxInteger (0,0 200x30), variable: varEnum, text list: 'TextListForCombobox_eReglertyp'
END_VISUALIZATION

// /VISU_HELPER_Combobox_eSignalform
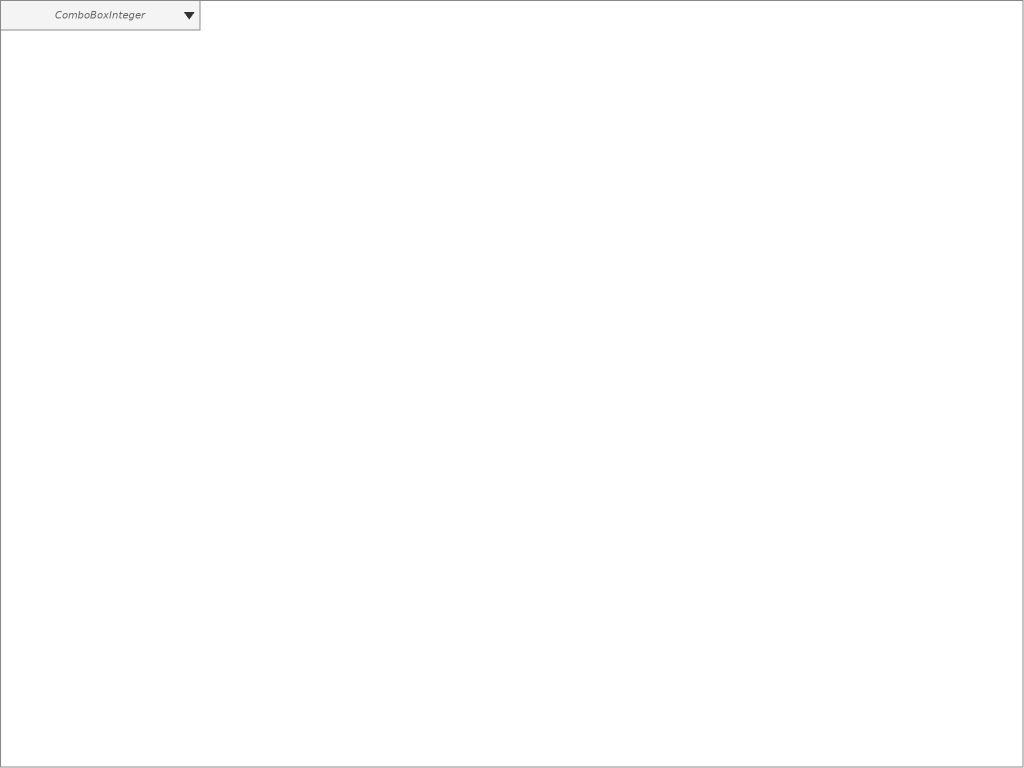
VISUALIZATION VISU_HELPER_Combobox_eSignalform  // 1024x768
VAR_IN_OUT
    varEnum : eSignalform;
END_VAR
    ComboBoxInteger (0,0 200x30), variable: varEnum, text list: 'TextListForCombobox_eSignalform'
END_VISUALIZATION

(* text list TextListForCombobox_eReglertyp (id | default)
  1 | P
  2 | I
  3 | PI
  4 | PDT1
  5 | PIDT1
   |  *)

(* text list TextListForCombobox_eSignalform (id | default)
  1 | OFF
  2 | OFFSET
  3 | RECHTECK
  4 | DREIECK
  5 | SINUS
  6 | RAMPE
   |  *)
